	// Arrayposition entspricht dem absoluten Druck. Z.B. 1.00bara => 0.00bar Überdruck => Arrayposition 100
	R407cDew: ARRAY [0..5100] OF INT := [-1006,-937,-894,-862,-835,-813,-794,-777,-762,-748,-735,-723,-712,-702,-692,-683,-674,-666,-658,-650,-643,-636,-629,-622,-616,-610,-604,-598,-593,-587,-582,-577,-572,-567,-562,-557,-553,-548,-544,-540,-535,-531,-527,-523,-519,-515,-512,-508,-504,-501,-497,-494,-490,-487,-484,-480,-477,-474,-471,-468,-465,-462,-459,-456,-453,-450,-447,-445,-442,-439,-436,-434,-431,-428,-426,-423,-421,-418,-416,-413,-411,-409,-406,-404,-402,-399,-397,-395,-392,-390,-388,-386,-384,-382,-379,-377,-375,-373,-371,-369,-367,-365,-363,-361,-359,-357,-355,-353,-351,-349,-347,-346,-344,-342,-340,-338,-336,-335,-333,-331,-329,-328,-326,-324,-322,-321,-319,-317,-316,-314,-312,-311,-309,-307,-306,-304,-303,-301,-300,-298,-296,-295,-293,-292,-290,-289,-287,-286,-284,-283,-281,-280,-278,-277,-275,-274,-273,-271,-270,-268,-267,-266,-264,-263,-261,-260,-259,-257,-256,-255,-253,-252,-251,-249,-248,-247,-245,-244,-243,-241,-240,-239,-238,-236,-235,-234,-233,-231,-230,-229,-228,-226,-225,-224,-223,-222,-220,-219,-218,-217,-216,-215,-213,-212,-211,-210,-209,-208,-206,-205,-204,-203,-202,-201,-200,-199,-197,-196,-195,-194,-193,-192,-191,-190,-189,-188,-187,-185,-184,-183,-182,-181,-180,-179,-178,-177,-176,-175,-174,-173,-172,-171,-170,-169,-168,-167,-166,-165,-164,-163,-162,-161,-160,-159,-158,-157,-156,-155,-154,-153,-152,-151,-150,-149,-148,-147,-146,-145,-145,-144,-143,-142,-141,-140,-139,-138,-137,-136,-135,-134,-133,-133,-132,-131,-130,-129,-128,-127,-126,-125,-124,-124,-123,-122,-121,-120,-119,-118,-118,-117,-116,-115,-114,-113,-112,-112,-111,-110,-109,-108,-107,-106,-106,-105,-104,-103,-102,-101,-101,-100,-99,-98,-97,-97,-96,-95,-94,-93,-93,-92,-91,-90,-89,-89,-88,-87,-86,-85,-85,-84,-83,-82,-81,-81,-80,-79,-78,-78,-77,-76,-75,-75,-74,-73,-72,-71,-71,-70,-69,-68,-68,-67,-66,-65,-65,-64,-63,-63,-62,-61,-60,-60,-59,-58,-57,-57,-56,-55,-55,-54,-53,-52,-52,-51,-50,-50,-49,-48,-47,-47,-46,-45,-45,-44,-43,-42,-42,-41,-40,-40,-39,-38,-38,-37,-36,-36,-35,-34,-34,-33,-32,-32,-31,-30,-29,-29,-28,-27,-27,-26,-25,-25,-24,-23,-23,-22,-22,-21,-20,-20,-19,-18,-18,-17,-16,-16,-15,-14,-14,-13,-12,-12,-11,-11,-10,-9,-9,-8,-7,-7,-6,-5,-5,-4,-4,-3,-2,-2,-1,0,0,1,1,2,3,3,4,4,5,6,6,7,8,8,9,9,10,11,11,12,12,13,14,14,15,15,16,17,17,18,18,19,20,20,21,21,22,22,23,24,24,25,25,26,27,27,28,28,29,29,30,31,31,32,32,33,33,34,35,35,36,36,37,37,38,38,39,40,40,41,41,42,42,43,43,44,45,45,46,46,47,47,48,48,49,50,50,51,51,52,52,53,53,54,54,55,55,56,57,57,58,58,59,59,60,60,61,61,62,62,63,63,64,64,65,66,66,67,67,68,68,69,69,70,70,71,71,72,72,73,73,74,74,75,75,76,76,77,77,78,78,79,79,80,80,81,81,82,82,83,83,84,84,85,85,86,86,87,87,88,88,89,89,90,90,91,91,92,92,93,93,94,94,95,95,96,96,97,97,98,98,99,99,100,100,101,101,101,102,102,103,103,104,104,105,105,106,106,107,107,108,108,109,109,110,110,110,111,111,112,112,113,113,114,114,115,115,116,116,117,117,117,118,118,119,119,120,120,121,121,122,122,122,123,123,124,124,125,125,126,126,127,127,127,128,128,129,129,130,130,131,131,131,132,132,133,133,134,134,135,135,135,136,136,137,137,138,138,139,139,139,140,140,141,141,142,142,142,143,143,144,144,145,145,145,146,146,147,147,148,148,148,149,149,150,150,151,151,151,152,152,153,153,154,154,154,155,155,156,156,156,157,157,158,158,159,159,159,160,160,161,161,161,162,162,163,163,164,164,164,165,165,166,166,166,167,167,168,168,168,169,169,170,170,170,171,171,172,172,173,173,173,174,174,175,175,175,176,176,177,177,177,178,178,179,179,179,180,180,181,181,181,182,182,182,183,183,184,184,184,185,185,186,186,186,187,187,188,188,188,189,189,190,190,190,191,191,191,192,192,193,193,193,194,194,195,195,195,196,196,196,197,197,198,198,198,199,199,199,200,200,201,201,201,202,202,203,203,203,204,204,204,205,205,206,206,206,207,207,207,208,208,209,209,209,210,210,210,211,211,211,212,212,213,213,213,214,214,214,215,215,216,216,216,217,217,217,218,218,218,219,219,220,220,220,221,221,221,222,222,222,223,223,223,224,224,225,225,225,226,226,226,227,227,227,228,228,228,229,229,230,230,230,231,231,231,232,232,232,233,233,233,234,234,234,235,235,236,236,236,237,237,237,238,238,238,239,239,239,240,240,240,241,241,241,242,242,242,243,243,244,244,244,245,245,245,246,246,246,247,247,247,248,248,248,249,249,249,250,250,250,251,251,251,252,252,252,253,253,253,254,254,254,255,255,255,256,256,256,257,257,257,258,258,258,259,259,259,260,260,260,261,261,261,262,262,262,263,263,263,264,264,264,265,265,265,266,266,266,267,267,267,268,268,268,269,269,269,270,270,270,271,271,271,272,272,272,272,273,273,273,274,274,274,275,275,275,276,276,276,277,277,277,278,278,278,279,279,279,280,280,280,280,281,281,281,282,282,282,283,283,283,284,284,284,285,285,285,286,286,286,286,287,287,287,288,288,288,289,289,289,290,290,290,291,291,291,291,292,292,292,293,293,293,294,294,294,295,295,295,295,296,296,296,297,297,297,298,298,298,299,299,299,299,300,300,300,301,301,301,302,302,302,302,303,303,303,304,304,304,305,305,305,305,306,306,306,307,307,307,308,308,308,308,309,309,309,310,310,310,311,311,311,311,312,312,312,313,313,313,314,314,314,314,315,315,315,316,316,316,316,317,317,317,318,318,318,319,319,319,319,320,320,320,321,321,321,321,322,322,322,323,323,323,323,324,324,324,325,325,325,325,326,326,326,327,327,327,328,328,328,328,329,329,329,330,330,330,330,331,331,331,332,332,332,332,333,333,333,334,334,334,334,335,335,335,335,336,336,336,337,337,337,337,338,338,338,339,339,339,339,340,340,340,341,341,341,341,342,342,342,342,343,343,343,344,344,344,344,345,345,345,346,346,346,346,347,347,347,347,348,348,348,349,349,349,349,350,350,350,350,351,351,351,352,352,352,352,353,353,353,353,354,354,354,355,355,355,355,356,356,356,356,357,357,357,358,358,358,358,359,359,359,359,360,360,360,361,361,361,361,362,362,362,362,363,363,363,363,364,364,364,365,365,365,365,366,366,366,366,367,367,367,367,368,368,368,368,369,369,369,370,370,370,370,371,371,371,371,372,372,372,372,373,373,373,373,374,374,374,375,375,375,375,376,376,376,376,377,377,377,377,378,378,378,378,379,379,379,379,380,380,380,380,381,381,381,382,382,382,382,383,383,383,383,384,384,384,384,385,385,385,385,386,386,386,386,387,387,387,387,388,388,388,388,389,389,389,389,390,390,390,390,391,391,391,391,392,392,392,392,393,393,393,393,394,394,394,394,395,395,395,395,396,396,396,396,397,397,397,397,398,398,398,398,399,399,399,399,400,400,400,400,401,401,401,401,402,402,402,402,403,403,403,403,404,404,404,404,405,405,405,405,406,406,406,406,407,407,407,407,408,408,408,408,409,409,409,409,409,410,410,410,410,411,411,411,411,412,412,412,412,413,413,413,413,414,414,414,414,415,415,415,415,416,416,416,416,416,417,417,417,417,418,418,418,418,419,419,419,419,420,420,420,420,421,421,421,421,421,422,422,422,422,423,423,423,423,424,424,424,424,425,425,425,425,426,426,426,426,426,427,427,427,427,428,428,428,428,429,429,429,429,429,430,430,430,430,431,431,431,431,432,432,432,432,433,433,433,433,433,434,434,434,434,435,435,435,435,436,436,436,436,436,437,437,437,437,438,438,438,438,439,439,439,439,439,440,440,440,440,441,441,441,441,441,442,442,442,442,443,443,443,443,444,444,444,444,444,445,445,445,445,446,446,446,446,446,447,447,447,447,448,448,448,448,449,449,449,449,449,450,450,450,450,451,451,451,451,451,452,452,452,452,453,453,453,453,453,454,454,454,454,455,455,455,455,455,456,456,456,456,457,457,457,457,457,458,458,458,458,459,459,459,459,459,460,460,460,460,461,461,461,461,461,462,462,462,462,462,463,463,463,463,464,464,464,464,464,465,465,465,465,466,466,466,466,466,467,467,467,467,467,468,468,468,468,469,469,469,469,469,470,470,470,470,471,471,471,471,471,472,472,472,472,472,473,473,473,473,474,474,474,474,474,475,475,475,475,475,476,476,476,476,477,477,477,477,477,478,478,478,478,478,479,479,479,479,479,480,480,480,480,481,481,481,481,481,482,482,482,482,482,483,483,483,483,484,484,484,484,484,485,485,485,485,485,486,486,486,486,486,487,487,487,487,487,488,488,488,488,489,489,489,489,489,490,490,490,490,490,491,491,491,491,491,492,492,492,492,492,493,493,493,493,493,494,494,494,494,495,495,495,495,495,496,496,496,496,496,497,497,497,497,497,498,498,498,498,498,499,499,499,499,499,500,500,500,500,500,501,501,501,501,501,502,502,502,502,502,503,503,503,503,504,504,504,504,504,505,505,505,505,505,506,506,506,506,506,507,507,507,507,507,508,508,508,508,508,509,509,509,509,509,510,510,510,510,510,511,511,511,511,511,512,512,512,512,512,513,513,513,513,513,514,514,514,514,514,515,515,515,515,515,515,516,516,516,516,516,517,517,517,517,517,518,518,518,518,518,519,519,519,519,519,520,520,520,520,520,521,521,521,521,521,522,522,522,522,522,523,523,523,523,523,524,524,524,524,524,525,525,525,525,525,525,526,526,526,526,526,527,527,527,527,527,528,528,528,528,528,529,529,529,529,529,530,530,530,530,530,530,531,531,531,531,531,532,532,532,532,532,533,533,533,533,533,534,534,534,534,534,535,535,535,535,535,535,536,536,536,536,536,537,537,537,537,537,538,538,538,538,538,539,539,539,539,539,539,540,540,540,540,540,541,541,541,541,541,542,542,542,542,542,542,543,543,543,543,543,544,544,544,544,544,545,545,545,545,545,545,546,546,546,546,546,547,547,547,547,547,548,548,548,548,548,548,549,549,549,549,549,550,550,550,550,550,550,551,551,551,551,551,552,552,552,552,552,553,553,553,553,553,553,554,554,554,554,554,555,555,555,555,555,555,556,556,556,556,556,557,557,557,557,557,557,558,558,558,558,558,559,559,559,559,559,559,560,560,560,560,560,561,561,561,561,561,561,562,562,562,562,562,563,563,563,563,563,563,564,564,564,564,564,565,565,565,565,565,565,566,566,566,566,566,567,567,567,567,567,567,568,568,568,568,568,568,569,569,569,569,569,570,570,570,570,570,570,571,571,571,571,571,572,572,572,572,572,572,573,573,573,573,573,573,574,574,574,574,574,575,575,575,575,575,575,576,576,576,576,576,576,577,577,577,577,577,578,578,578,578,578,578,579,579,579,579,579,579,580,580,580,580,580,580,581,581,581,581,581,582,582,582,582,582,582,583,583,583,583,583,583,584,584,584,584,584,585,585,585,585,585,585,586,586,586,586,586,586,587,587,587,587,587,587,588,588,588,588,588,588,589,589,589,589,589,590,590,590,590,590,590,591,591,591,591,591,591,592,592,592,592,592,592,593,593,593,593,593,593,594,594,594,594,594,594,595,595,595,595,595,595,596,596,596,596,596,597,597,597,597,597,597,598,598,598,598,598,598,599,599,599,599,599,599,600,600,600,600,600,600,601,601,601,601,601,601,602,602,602,602,602,602,603,603,603,603,603,603,604,604,604,604,604,604,605,605,605,605,605,605,606,606,606,606,606,606,607,607,607,607,607,607,608,608,608,608,608,608,609,609,609,609,609,609,610,610,610,610,610,610,611,611,611,611,611,611,612,612,612,612,612,612,613,613,613,613,613,613,614,614,614,614,614,614,615,615,615,615,615,615,615,616,616,616,616,616,616,617,617,617,617,617,617,618,618,618,618,618,618,619,619,619,619,619,619,620,620,620,620,620,620,621,621,621,621,621,621,622,622,622,622,622,622,622,623,623,623,623,623,623,624,624,624,624,624,624,625,625,625,625,625,625,626,626,626,626,626,626,627,627,627,627,627,627,627,628,628,628,628,628,628,629,629,629,629,629,629,630,630,630,630,630,630,630,631,631,631,631,631,631,632,632,632,632,632,632,633,633,633,633,633,633,634,634,634,634,634,634,634,635,635,635,635,635,635,636,636,636,636,636,636,637,637,637,637,637,637,637,638,638,638,638,638,638,639,639,639,639,639,639,639,640,640,640,640,640,640,641,641,641,641,641,641,642,642,642,642,642,642,642,643,643,643,643,643,643,644,644,644,644,644,644,644,645,645,645,645,645,645,646,646,646,646,646,646,646,647,647,647,647,647,647,648,648,648,648,648,648,648,649,649,649,649,649,649,650,650,650,650,650,650,650,651,651,651,651,651,651,652,652,652,652,652,652,652,653,653,653,653,653,653,654,654,654,654,654,654,654,655,655,655,655,655,655,655,656,656,656,656,656,656,657,657,657,657,657,657,657,658,658,658,658,658,658,659,659,659,659,659,659,659,660,660,660,660,660,660,660,661,661,661,661,661,661,662,662,662,662,662,662,662,663,663,663,663,663,663,663,664,664,664,664,664,664,665,665,665,665,665,665,665,666,666,666,666,666,666,666,667,667,667,667,667,667,667,668,668,668,668,668,668,669,669,669,669,669,669,669,670,670,670,670,670,670,670,671,671,671,671,671,671,671,672,672,672,672,672,672,673,673,673,673,673,673,673,674,674,674,674,674,674,674,675,675,675,675,675,675,675,676,676,676,676,676,676,676,677,677,677,677,677,677,677,678,678,678,678,678,678,678,679,679,679,679,679,679,680,680,680,680,680,680,680,681,681,681,681,681,681,681,682,682,682,682,682,682,682,683,683,683,683,683,683,683,684,684,684,684,684,684,684,685,685,685,685,685,685,685,686,686,686,686,686,686,686,687,687,687,687,687,687,687,688,688,688,688,688,688,688,689,689,689,689,689,689,689,690,690,690,690,690,690,690,691,691,691,691,691,691,691,692,692,692,692,692,692,692,693,693,693,693,693,693,693,694,694,694,694,694,694,694,695,695,695,695,695,695,695,695,696,696,696,696,696,696,696,697,697,697,697,697,697,697,698,698,698,698,698,698,698,699,699,699,699,699,699,699,700,700,700,700,700,700,700,701,701,701,701,701,701,701,701,702,702,702,702,702,702,702,703,703,703,703,703,703,703,704,704,704,704,704,704,704,705,705,705,705,705,705,705,705,706,706,706,706,706,706,706,707,707,707,707,707,707,707,708,708,708,708,708,708,708,709,709,709,709,709,709,709,709,710,710,710,710,710,710,710,711,711,711,711,711,711,711,712,712,712,712,712,712,712,712,713,713,713,713,713,713,713,714,714,714,714,714,714,714,715,715,715,715,715,715,715,715,716,716,716,716,716,716,716,717,717,717,717,717,717,717,717,718,718,718,718,718,718,718,719,719,719,719,719,719,719,719,720,720,720,720,720,720,720,721,721,721,721,721,721,721,721,722,722,722,722,722,722,722,723,723,723,723,723,723,723,723,724,724,724,724,724,724,724,725,725,725,725,725,725,725,725,726,726,726,726,726,726,726,727,727,727,727,727,727,727,727,728,728,728,728,728,728,728,729,729,729,729,729,729,729,729,730,730,730,730,730,730,730,730,731,731,731,731,731,731,731,732,732,732,732,732,732,732,732,733,733,733,733,733,733,733,733,734,734,734,734,734,734,734,735,735,735,735,735,735,735,735,736,736,736,736,736,736,736,736,737,737,737,737,737,737,737,738,738,738,738,738,738,738,738,739,739,739,739,739,739,739,739,740,740,740,740,740,740,740,740,741,741,741,741,741,741,741,741,742,742,742,742,742,742,742,743,743,743,743,743,743,743,743,744,744,744,744,744,744,744,744,745,745,745,745,745,745,745,745,746,746,746,746,746,746,746,746,747,747,747,747,747,747,747,747,748,748,748,748,748,748,748,748,749,749,749,749,749,749,749,749,750,750,750,750,750,750,750,750,751,751,751,751,751,751,751,752,752,752,752,752,752,752,752,753,753,753,753,753,753,753,753,754,754,754,754,754,754,754,754,755,755,755,755,755,755,755,755,755,756,756,756,756,756,756,756,756,757,757,757,757,757,757,757,757,758,758,758,758,758,758,758,758,759,759,759,759,759,759,759,759,760,760,760,760,760,760,760,760,761,761,761,761,761,761,761,761,762,762,762,762,762,762,762,762,763,763,763,763,763,763,763,763,764,764,764,764,764,764,764,764,764,765,765,765,765,765,765,765,765,766,766,766,766,766,766,766,766,767,767,767,767,767,767,767,767,768,768,768,768,768,768,768,768,768,769,769,769,769,769,769,769,769,770,770,770,770,770,770,770,770,771,771,771,771,771,771,771,771,771,772,772,772,772,772,772,772,772,773,773,773,773,773,773,773,773,774,774,774,774,774,774,774,774,774,775,775,775,775,775,775,775,775,776,776,776,776,776,776,776,776,777,777,777,777,777,777,777,777,777,778,778,778,778,778,778,778,778,779,779,779,779,779,779,779,779,779,780,780,780,780,780,780,780,780,781,781,781,781,781,781,781,781,781,782,782,782,782,782,782,782,782,783,783,783,783,783,783,783,783,783,784,784,784,784,784,784,784,784,784,785,785,785,785,785,785,785,785,786,786,786,786,786,786,786,786,786,787,787,787,787,787,787,787,787,788,788,788,788,788,788,788,788,788,789,789,789,789,789,789,789,789,789,790,790,790,790,790,790,790,790,791,791,791,791,791,791,791,791,791,792,792,792,792,792,792,792,792,792,793,793,793,793,793,793,793,793,793,794,794,794,794,794,794,794,794,795,795,795,795,795,795,795,795,795,796,796,796,796,796,796,796,796,796,797,797,797,797,797,797,797,797,797,798,798,798,798,798,798,798,798,798,799,799,799,799,799,799,799,799,799,800,800,800,800,800,800,800,800,800,801,801,801,801,801,801,801,801,801,802,802,802,802,802,802,802,802,802,803,803,803,803,803,803,803,803,803,804,804,804,804,804,804,804,804,804,805,805,805,805,805,805,805,805,805,806,806,806,806,806,806,806,806,806,807,807,807,807,807,807,807,807,807,808,808,808,808,808,808,808,808,808,809,809,809,809,809,809,809,809,809,810,810,810,810,810,810,810,810,810,811,811,811,811,811,811,811,811,811,811,812,812,812,812,812,812,812,812,812,813,813,813,813,813,813,813,813,813,814,814,814,814,814,814,814,814,814,815,815,815,815,815,815,815,815,815,815,816,816,816,816,816,816,816,816,816,817,817,817,817,817,817,817,817,817,818,818,818,818,818,818,818,818,818,818,819,819,819,819,819,819,819,819,819,820,820,820,820,820,820,820,820,820,820,821,821,821,821,821,821,821,821,821,822,822,822,822,822,822,822,822,822,822,823,823,823,823,823,823,823,823,823,824,824];

END_VAR

// Globale Variablen/SW_ALZ
{attribute 'qualified_only'}
VAR_GLOBAL
	Bitzer_Scroll_R410a: SW_Einsatzgrenzen := (f_SW_EG_MinVerd := -30, f_SW_EG_MaxVerd := 21, f_SW_EG_MinKond := 25, f_SW_EG_MaxKond := 65, f_SW_EG_BVerd := 12.5, f_SW_EG_BKond := 25, f_SW_EG_CKond := 38, f_SW_EG_DKond := 65, f_SW_EG_EVerd := 21, f_SW_EG_FVerd := 0, f_SW_EG_GKond := 32, f_SW_Max_HeissgasTemp := 120);
END_VAR

// Globale Variablen/Visu
{attribute 'qualified_only'}
VAR_GLOBAL
	i_Frame_Index:INT;
	i_Verschiebung_Horizontal:INT;
	i_Verschiebung_Vertikal:INT;
	x_Quittieren: BOOL;
END_VAR

// Version/Global_Version
{attribute 'TcGenerated'}
// This function has been automatically generated from the project information.
VAR_GLOBAL CONSTANT
	{attribute 'const_non_replaced'}
	{attribute 'linkalways'}
	stLibVersion_GWP_Library : ST_LibVersion := (iMajor := 17, iMinor := 9, iBuild := 1, iRevision := 0, sVersion := '17.9.1');
END_VAR

// Allgemein/Alarm
(*Alarmblock, welcher ein digitaler Ausgang high setzt wenn mind. Ein Alarm anstehend ist und ebenfalls noch die Selbsthaltung der Alarme
*)
FUNCTION_BLOCK Alarm
(*
Versionsverlauf: 
Version		|Autor	|Bemerkung
------------------------------------------------------------------------------------------------------------ 
17.06.00	|Shgb	|erste Freigabe 
17.08.00	|LeaF	|Freigabe

*)
VAR_INPUT
	x_AL1:BOOL;//Alarmeingang 1-16
	x_AL2:BOOL;
	x_AL3:BOOL;
	x_AL4:BOOL;
	x_AL5:BOOL;
	x_AL6:BOOL;
	x_AL7:BOOL;
	x_AL8:BOOL;
	x_AL9:BOOL;
	x_AL10:BOOL;
END_VAR
VAR_OUTPUT	
	x_Aus:BOOL;//Allgemeiner Alarm
	x_AL_1:BOOL;//Alarmausgang 1-16
	x_AL_2:BOOL;
	x_AL_3:BOOL;
	x_AL_4:BOOL;
	x_AL_5:BOOL;
	x_AL_6:BOOL;
	x_AL_7:BOOL;
	x_AL_8:BOOL;
	x_AL_9:BOOL;
	x_AL_10:BOOL;
END_VAR
VAR Persistent
	ax_AL :ARRAY [1..10] OF BOOL;
	ax_Speicher :ARRAY [1..10] OF BOOL;
	i_Arraypos:INT;
	as_Liste: ARRAY [1..10] OF STRING;
END_VAR

//Array füllen
	ax_AL[1]:=x_AL1;
	ax_AL[2]:=x_AL2;
	ax_AL[3]:=x_AL3;
	ax_AL[4]:=x_AL4;
	ax_AL[5]:=x_AL5;
	ax_AL[6]:=x_AL6;
	ax_AL[7]:=x_AL7;
	ax_AL[8]:=x_AL8;
	ax_AL[9]:=x_AL9;
	ax_AL[10]:=x_AL10;
	
//Quittieren
	IF Globale_Variablen.x_Quittieren THEN
		FOR i_Arraypos:=1 TO 10 DO
			ax_Speicher[i_Arraypos]:=FALSE;
		END_FOR
	END_IF

//Alarme Setzen
	FOR i_Arraypos:=1 TO 10 DO
		IF ax_AL[i_Arraypos] THEN
			ax_Speicher[i_Arraypos]:=TRUE;
		END_IF
	END_FOR

//Ausgäne setzen
	x_AL_1:=ax_Speicher[1];
	x_AL_2:=ax_Speicher[2];
	x_AL_3:=ax_Speicher[3];
	x_AL_4:=ax_Speicher[4];
	x_AL_5:=ax_Speicher[5];
	x_AL_6:=ax_Speicher[6];
	x_AL_7:=ax_Speicher[7];
	x_AL_8:=ax_Speicher[8];
	x_AL_9:=ax_Speicher[9];
	x_AL_10:=ax_Speicher[10];
	
	x_Aus:=x_al_1 OR 
			x_al_2 OR 
			x_al_3 OR 
			x_al_4 OR
			x_al_5 OR
			x_al_6 OR
			x_al_7 OR
			x_al_8 OR
			x_al_9 OR
			x_al_10;

END_FUNCTION_BLOCK

// Allgemein/COUNT
(*Je nachdem wieviele digitale Eingänge true sind, wird er analoge Ausgang hochgezählt. Ist kein Eingang auf true, bleibt der Ausgang auf 0.
Der Counter ist auf max. 8 digitale Eingänge ausgelegt.
*)
FUNCTION_BLOCK COUNT
(*
Versionsverlauf: 
Version		|Autor	|Bemerkung
------------------------------------------------------------------------------------------------------------ 
17.05.00	|KuzR	|erste Freigabe  
17.08.00	|LeaF	|Freigabe

*)
VAR_INPUT	
	x_Ein_1:BOOL;//8 Digitale Eingänge
	x_Ein_2:BOOL;
	x_Ein_3:BOOL;
	x_Ein_4:BOOL;
	x_Ein_5:BOOL;
	x_Ein_6:BOOL;
	x_Ein_7:BOOL;
	x_Ein_8:BOOL;
END_VAR
VAR_OUTPUT
	i_Aus:Int;//Ausganng in Int
END_VAR
VAR	
END_VAR

	i_Aus:=0;
// Ausgang zählt hoch, wenn Eingang true ist
	IF x_Ein_1 THEN
		i_Aus:=i_Aus+1;
	END_IF
	
	IF x_Ein_2 THEN
		i_Aus:=i_Aus+1;
	END_IF
	
	IF x_Ein_3 THEN
		i_Aus:=i_Aus+1;
	END_IF
	
	IF x_Ein_4 THEN
		i_Aus:=i_Aus+1;
	END_IF
	
	IF x_Ein_5 THEN
		i_Aus:=i_Aus+1;
	END_IF
	
	IF x_Ein_6 THEN
		i_Aus:=i_Aus+1;
	END_IF
	
	IF x_Ein_7 THEN
		i_Aus:=i_Aus+1;
	END_IF
	
	IF x_Ein_8 THEN
		i_Aus:=i_Aus+1;
	END_IF

END_FUNCTION_BLOCK

// Allgemein/MUX_B
(*Anhand von 4 digitalen Eingängen wird entschieden, welcher von 4 analogen Werten (Real) auf den analogen Ausgang (Real) geschrieben wird.
Der kleinere Eingang hat immer Priorität für das Schreiben des Ausganges. Wenn keine Eingänge auf true sind, dann Augang auf 0.

*)
FUNCTION_BLOCK MUX_B
(*
Versionsverlauf: 
Version		|Autor	|Bemerkung
------------------------------------------------------------------------------------------------------------ 
17.06.00	|KuzR	|erste Freigabe  
17.08.00	|LeaF	|Freigabe

*)
VAR_INPUT
	f_Ein_1:REAL;//Eingangswerte 1-4 in Real
	f_Ein_2:REAL;
	f_Ein_3:REAL;
	f_Ein_4:REAL;
	x_Ein_1:BOOL;//Digitaler Eingang 1
	x_Ein_2:BOOL;//Digitaler Eingang 2
	x_Ein_3:BOOL;//Digitaler Eingang 3
	x_Ein_4:BOOL;//Digitaler Eingang 4
END_VAR
VAR_OUTPUT
	f_Aus:REAL;//Ausgang in Real
END_VAR
VAR
END_VAR

	f_Aus:=0;
//Wenn 1.Eingang True, dann Wert1
	IF x_Ein_1  THEN
		f_Aus := f_Ein_1;		
//Ansonsen wird beim Ausgang Wert zwei geschrieben
	ELSIF x_Ein_2 THEN
		f_Aus := f_Ein_2;		
	ELSIF x_Ein_3 THEN
		f_Aus := f_Ein_3;		
	ELSIF x_Ein_4 THEN
		f_Aus := f_Ein_4;							
	END_IF

END_FUNCTION_BLOCK

// Allgemein/MUX_D_INT
(*Anhand von 3 analogen Eingangswerten (Integer)wird mit dem i_Sel entschieden, welcher von den 3 Eingängen auf den analogen Ausgang (Integer) geschrieben wird.
*)
FUNCTION_BLOCK MUX_D_INT
(*
Versionsverlauf: 
Version		|Autor	|Bemerkung
------------------------------------------------------------------------------------------------------------ 
17.05.00	|KuzR	|erste Freigabe  
17.08.00	|LeaF	|Freigabe

*)
VAR_INPUT
	i_Ein_1:INT;//Eingangswert 1 als Int
	i_Ein_2:INT;//Eingangswert 2 als Int
	i_Ein_3:INT; //Eingangswert 3 als Int
	i_Sel:INT;// Auswahl Selector
	
END_VAR
VAR_OUTPUT
	i_Aus:INT;//Ausgang als Int
END_VAR
VAR
END_VAR

//Mit Select Auswählen, welcher Eingang auf Ausgang geschrieben wird
	CASE i_sel OF
		1: i_Aus:= i_Ein_1;
		2: i_Aus:= i_Ein_2;
		3: i_Aus:= i_Ein_3;
	ELSE	
//Wenn Select <3 oder >0, dann Ausgang 0
		i_Aus:=0;
	END_CASE

END_FUNCTION_BLOCK

// Allgemein/MUX_D_REAL
(*Anhand von 3 analogen Eingangswerten (Real)wird mit dem i_Sel entschieden, welcher von den 3 Eingängen auf den analogen Ausgang (Real) geschrieben wird.
*)
FUNCTION_BLOCK MUX_D_REAL
(*
Versionsverlauf: 
Version		|Autor	|Bemerkung
------------------------------------------------------------------------------------------------------------ 
17.06.00	|ShgB	|erste Freigabe  
17.08.00	|LeaF	|Freigabe

*)
VAR_INPUT
	f_Ein_1:REAL;//Eingangswert 1 als Real
	f_Ein_2:REAL;//Eingangswert 2 als Real
	f_Ein_3:REAL;//Eingangswert 3 als Real
	i_Sel:INT;// Auswahl Selector
	
END_VAR
VAR_OUTPUT
	f_Aus:REAL;//Ausgang in Real
END_VAR
VAR
END_VAR

//Mit Select Auswählen, welcher Eingang auf Ausgang geschrieben wird
	CASE i_sel OF
		1: f_Aus:= f_Ein_1;
		2: f_Aus:= f_Ein_2;
		3: f_Aus:= f_Ein_3;
	ELSE
		
//Wenn Select <0 oder >3, dann Ausgang 0
		f_Aus:=0;
	END_CASE

END_FUNCTION_BLOCK

// Allgemein/NULL
(*Wenn der analoge Eingang (Real) genau 0 ist, wird der digitale Ausgang auf true gesetzt, ansonsten auf false.
*)
FUNCTION_BLOCK NULL
(*
Versionsverlauf: 
Version		|Autor	|Bemerkung
------------------------------------------------------------------------------------------------------------ 
17.06.00	|KuzR	|erste Freigabe  
17.08.00	|LeaF	|Freigabe

*)
VAR_INPUT
	i_Ein:REAL;//Eingangswert in Real
END_VAR
VAR_OUTPUT
	x_Aus:BOOL;//Digitaler Ausgang
END_VAR
VAR
END_VAR

//Wenn 0 gleich Ausgang true, ansonsten false
	x_Aus:=i_Ein =0;

END_FUNCTION_BLOCK

// Allgemein/SWITCH_INT
(*Ist der digitale Eingang auf false, wird der erste analoge Eingangswert (Int) in den analogen Ausgang (Int) geschrieben. 
Ist der digitale Eingang auf true, wird der zweite analoge Eingangswert (Int) in den analogen Ausgang (Int) geschrieben.
*)
FUNCTION_BLOCK SWITCH_INT
(*
Versionsverlauf: 
Version		|Autor	|Bemerkung
------------------------------------------------------------------------------------------------------------ 
17.05.00	|KuzR	|erste Freigabe  
17.08.00	|LeaF	|Freigabe

*)
VAR_INPUT
	x_Ein:BOOL;//Digitaler Eingang
	i_Ein_1:INT;//Analoger Eingangswert 1 als Int
	i_Ein_2:INT;//Analoger Eingangswert 2 als Int
END_VAR
VAR_OUTPUT
	i_Aus:INT;//Analoger Ausgangswert als Int
END_VAR
VAR	
END_VAR

	IF x_Ein THEN		
//Wenn Eingang True, Wert_2 in Ausgang
		i_Aus:= i_Ein_2;	
	ELSE	
//Wenn Eingang false, Wert_1 in Ausgang
		i_Aus:= i_Ein_1;
	END_IF

END_FUNCTION_BLOCK

// Allgemein/SWITCH_REAL
(*Ist der digitale Eingang auf false, wird der erste analoge Eingangswert (Real) in den analogen Ausgang (Real) geschrieben. 
Ist der digitale Eingang auf true, wird der zweite analoge Eingangswert (Real) in den analogen Ausgang (Real) geschrieben.
*)
FUNCTION_BLOCK SWITCH_REAL
(*
Versionsverlauf: 
Version		|Autor	|Bemerkung
------------------------------------------------------------------------------------------------------------ 
17.05.00	|KuzR	|erste Freigabe  
17.08.00	|LeaF	|Freigabe

*)
VAR_INPUT
	x_Ein:BOOL;//Digitaler Eingang
	f_Ein_1:REAL;//Analoger Eingangswert 1 als Real
	f_Ein_2	:REAL;//Analoger Eingangswert 2 als Real
END_VAR
VAR_OUTPUT
	f_Aus:REAL;//Analoger Ausgangswert als Real
END_VAR
VAR	
END_VAR

	IF x_Ein THEN		
//Wenn Eingang True, Wert_2 in Ausgang
		f_Aus:= f_Ein_2;	
	ELSE	
//Wenn Eingang false, Wert_1 in Ausgang
		f_Aus:= f_Ein_1;
	END_IF

END_FUNCTION_BLOCK

// Allgemein/Toggle
(*Mit einer positiven Flanke auf den x_Toggle Eingang wird der Wert des Ausgangs x_Aus zwischen FALSE und TRUE gwechselt.
Mit dem x_Reset Eingang kann der Ausgang auf FALSE geschrieben werden. 
*)
FUNCTION_BLOCK Toggle
(*
Versionsverlauf: 
Version		|Autor	|Bemerkung
------------------------------------------------------------------------------------------------------------ 
17.06.00	|Shgb	|erste Freigabe  
17.08.00	|LeaF	|Freigabe

*)
VAR_INPUT
	x_Toggle:BOOL;//Wechselt den Wert des Ausgangs bei einer positiven Flanke
	x_Reset:BOOL;//Setzt den Ausgang auf FALSE
END_VAR
VAR_OUTPUT
	x_Aus:BOOL;//Ausgang
END_VAR
VAR PERSISTENT
	x_Speicher: BOOL;
END_VAR
VAR
	x_Flanke:BOOL;
END_VAR

//Toggle mit Flankenerkennung
	IF x_Toggle AND NOT x_Flanke THEN
		x_Speicher:= NOT x_Speicher;
	END_IF
	x_Flanke:=x_Toggle;

//Reset
	IF x_Reset THEN
		x_Speicher:=FALSE;
	END_IF
	
//Ausgang schreiben
	x_Aus:=x_Speicher;

END_FUNCTION_BLOCK

// Converters/Converter2Punkt
(*Der Eingang f_Ein wird anhand des Bereiches von f_Ein_Min f_Ein_Max auf den Bereich f_Aus_Min und f_Aus_Max berechnet und auf den Ausgang f_Aus gegeben.
*)
FUNCTION_BLOCK Converter2Punkt
(*
Versionsverlauf: 
Version		|Autor	|Bemerkung
------------------------------------------------------------------------------------------------------------ 
17.06.00	|ShgB	|erste Freigabe 
17.06.01	|ShgB	|von Integer auf Real geändert 
17.08.00	|LeaF	|Freigabe	

*)
VAR_INPUT
	f_Ein:REAL;//Eingang
	f_Ein_Min:REAL;//Eingangsbereich Minimum
	f_Ein_Max:REAL;//Eingangsbereich Maximum
	f_Aus_Min:REAL;//Ausgangsbereich Minimum
	f_Aus_Max:REAL;//Ausgangsbereich Maximum
END_VAR
VAR_OUTPUT
	f_Aus:REAL;//Ausgang
END_VAR
VAR
END_VAR

IF f_Ein_Max-f_Ein_Min <> 0 THEN
	f_Aus:=(f_Aus_Max-f_Aus_Min)/(f_Ein_Max-f_Ein_Min)*(f_Ein-f_Ein_Min)+f_Aus_Min;
ELSE
	f_Aus:=f_Aus_Max;
END_IF

END_FUNCTION_BLOCK

// Math/Maximum
(*Gibt den grössten der angeschlossenen Werten aus.
*)
FUNCTION_BLOCK Maximum
(*
Versionsverlauf: 
Version		|Autor	|Bemerkung
------------------------------------------------------------------------------------------------------------ 
17.06.00	|Shgb	|erste Freigabe 
17.06.01	|ShgB	|von Integer auf Real geändert	 
17.08.00	|LeaF	|Freigabe

*)
VAR_INPUT
	f_Ein1 :REAL:=0.00001;//Wert 1
	f_Ein2 :REAL:=0.00001;//Wert 2
	f_Ein3 :REAL:=0.00001;//Wert 3
	f_Ein4 :REAL:=0.00001;//Wert 4
	f_Ein5 :REAL:=0.00001;//Wert 5
	f_Ein6 :REAL:=0.00001;//Wert 6
	f_Ein7 :REAL:=0.00001;//Wert 7
	f_Ein8 :REAL:=0.00001;//Wert 8
END_VAR
VAR_OUTPUT
	f_Aus:REAL;//Grösste Wert
END_VAR
VAR
	i_Arraypos:INT;
	af_Array: ARRAY [1..8] OF REAL;
END_VAR

// Werte in Array platzieren
	af_Array[1]:=f_Ein1;
	af_Array[2]:=f_Ein2;
	af_Array[3]:=f_Ein3;
	af_Array[4]:=f_Ein4;
	af_Array[5]:=f_Ein5;
	af_Array[6]:=f_Ein6;
	af_Array[7]:=f_Ein7;
	af_Array[8]:=f_Ein8;
	
//Zahlen die kleiner als 0 sind
	f_Aus := af_Array[1];	
	
//Auswertung der grössten Zahl
	FOR i_Arraypos:=2 TO 8 DO
		IF af_Array[i_Arraypos] >= f_Aus AND af_Array[i_Arraypos] <> 0.00001 THEN
			f_Aus := af_Array[i_Arraypos];
		END_IF
	END_FOR

END_FUNCTION_BLOCK

// Converters/Int_to_Druck
(*Der analoge Wert der Eingangskarte wird von einem 16 bit Integer in einen REAL Wert umgewandelt und ein Offset dazu addiert.
Standardmässig ist der Eingangsbereich von 0 - 32767 eingestellt. Sollte dieser nicht übereinstimmen kann der Bereich angepasst werden.
*)
FUNCTION_BLOCK Int_to_Druck
(*
Versionsverlauf: 
Version		|Autor	|Bemerkung
------------------------------------------------------------------------------------------------------------ 
17.06.00	|Shgb	|erste Freigabe  
17.08.00	|LeaF	|Freigabe

*)
VAR_INPUT
	i_Ein:INT;//Digitaler Eingangswert
END_VAR
VAR_INPUT PERSISTENT
	i_Ein_Min:INT:=0;//Eingangsbereich Minimum
	i_Ein_Max:INT:=32767;//Eingangsbereich Maximum
	f_Aus_Min:REAL;//Minimum des Drucktransmitters
	f_Aus_Max:REAL;//Maximum des Drucktransmitters
	f_Offset:REAL;//Offset der dazu addiert wird
END_VAR
VAR_OUTPUT
	f_Aus:REAL;//Druck im REAL Format
END_VAR
VAR//GUI Variablen
	f_GUI_Input:REAL;
END_VAR

IF i_Ein_Max-i_Ein_Min <> 0 THEN
	f_Aus:=(f_Aus_Max-f_Aus_Min)/(i_Ein_Max-i_Ein_Min)*(i_Ein-i_Ein_Min)+f_Aus_Min+f_Offset;
ELSE
	f_Aus:=f_Aus_Min;
END_IF

f_GUI_Input:=f_Aus-f_Offset;

END_FUNCTION_BLOCK

// Converters/Int_to_Temperature
(*Wandelt die Temperatur im INT Format, die von der Eingangskarte kommt, in eine Temperatur in REAL Format um und rechnet einen Offset dazu.
*)
FUNCTION_BLOCK Int_to_Temperature
(*
Versionsverlauf: 
Version		|Autor	|Bemerkung
------------------------------------------------------------------------------------------------------------ 
17.06.00	|Shgb	|erste Freigabe  
17.08.00	|LeaF	|Freigabe

*)
VAR_INPUT
	i_Ein:INT;//Temperatur von Karte
END_VAR
VAR_INPUT PERSISTENT
	f_Offset:REAL;//Offset der dazu addiert wird
END_VAR
VAR_OUTPUT
	f_Temperatur:REAL;//Ausgang REAL
END_VAR
VAR//GUI Variablen
	f_GUI_Input:REAL;
END_VAR

f_Temperatur:=i_Ein/10.0+f_Offset;
f_GUI_Input:=i_Ein/10.0;

END_FUNCTION_BLOCK

// Converters/Prozent_to_Int
(*Wandelt eine Prozentangabe vom Format REAL in eine Integer Zahl für die analoge Augangskarte um.
Standardmässig ist der Eingangsbereich von 0 - 32767 eingestellt. Sollte dieser nicht übereinstimmen kann der Bereich angepasst werden.
*)
FUNCTION_BLOCK Prozent_to_Int
(*
Versionsverlauf: 
Version		|Autor	|Bemerkung
------------------------------------------------------------------------------------------------------------ 
17.06.00	|Shgb	|erste Freigabe 
17.08.00	|LeaF	|Freigabe 

*)
VAR_INPUT
	f_Ein:REAL;//Eingang in Prozent
END_VAR
VAR_INPUT PERSISTENT
	i_Aus_Min:INT:=0;//Eingangsbereich Minimum
	i_Aus_Max:INT:=32767;//eingangsbereich Maximum
END_VAR
VAR_OUTPUT
	f_Aus:INT;//Ausgang
END_VAR
VAR
END_VAR

f_Aus:=real_to_int((i_Aus_Max-i_Aus_Min)*f_Ein/100.0);

END_FUNCTION_BLOCK

// Converters/Time_to_Timestruct
(*Wandelt die Eingangsvariable vom Typ TIME in ein TIMESTRUCT um.
*)
FUNCTION_BLOCK Time_to_Timestruct
(*
Versionsverlauf: 
Version		|Autor	|Bemerkung
------------------------------------------------------------------------------------------------------------ 
17.06.00	|Shgb	|erste Freigabe 	 
17.08.00	|LeaF	|Freigabe

*)
VAR_INPUT
	t_Ein:TIME;//Eingang
END_VAR
VAR_OUTPUT
	t_Aus:timestruct;//Ausgang
END_VAR
VAR
	OT:OTSTRUCT;
END_VAR

OT:=TIME_TO_OTSTRUCT(t_Ein);
t_Aus.wMilliseconds:=ot.wMilliseconds;
t_Aus.wSecond:=ot.wSecond;
t_Aus.wMinute:=ot.wMinute;
t_Aus.wHour:=ot.wHour;
t_Aus.wDay:=ot.wDay+ot.wWeek*7;

END_FUNCTION_BLOCK

// Converters/Timestruct_to_Time
(*Wandelt einen TIMESTRUCT in die Ausgangsvariable vom Typ TIME um.
*)
FUNCTION_BLOCK Timestruct_to_Time
(*
Versionsverlauf: 
Version		|Autor	|Bemerkung
------------------------------------------------------------------------------------------------------------ 
17.06.00	|Shgb	|erste Freigabe  
17.08.00	|LeaF	|Freigabe	

*)
VAR_INPUT
	t_Ein:timestruct;//Eingang
END_VAR
VAR_OUTPUT
	t_Aus:TIME;//Ausgang
END_VAR
VAR
END_VAR

t_Aus:=DINT_TO_TIME(t_Ein.wMilliseconds
					+ t_Ein.wSecond*1000
					+ t_Ein.wMinute*1000*60
					+ t_Ein.wHour*1000*60*60
					+ t_Ein.wDay*1000*60*60*24);

END_FUNCTION_BLOCK

// Druck_Temp/R1234ze
(*Wandelt den Druck in die Entsprechende Temperatur um. Die Druck-Temperatur Werte sind in der Nassdampftabelle in den Globalen Variablen hinterlegt.
*)
FUNCTION_BLOCK R1234ze
(*
Versionsverlauf: 
Version		|Autor	|Bemerkung
------------------------------------------------------------------------------------------------------------ 
17.06.00	|Shgb	|erste Freigabe 
17.06.01	|ShgB	|von Integer auf Real geändert	 
17.08.00	|LeaF	|Freigabe

*)
VAR_INPUT
	f_ND:REAL;//Druck für Verdampfungstemperatur
	f_HD:REAL;//Druck für Kondensationstemperatur
END_VAR
VAR_OUTPUT
	f_VerdTemp:REAL;//Verdampfungstemperatur
	f_KondTemp:REAL;//Kondensationstemperatur
END_VAR
VAR
END_VAR

//Niederdruck
	f_VerdTemp:=Nassdampftabelle.R1234ze[REAL_TO_INT(f_ND*100)+100]/10.0;
	
//Hochdruck
	f_KondTemp:=Nassdampftabelle.R1234ze[REAL_TO_INT(f_HD*100)+100]/10.0;

END_FUNCTION_BLOCK

// Druck_Temp/R134a
(*Wandelt den Druck in die Entsprechende Temperatur um. Die Druck-Temperatur Werte sind in der Nassdampftabelle in den Globalen Variablen hinterlegt.
*)
FUNCTION_BLOCK R134a
(*
Versionsverlauf: 
Version		|Autor	|Bemerkung
------------------------------------------------------------------------------------------------------------ 
17.06.00	|Shgb	|erste Freigabe 
17.06.01	|ShgB	|von Integer auf Real geändert	 
17.08.00	|LeaF	|Freigabe

*)
VAR_INPUT
	f_ND:REAL;//Druck für Verdampfungstemperatur
	f_HD:REAL;//Druck für Kondensationstemperatur
END_VAR
VAR_OUTPUT
	f_VerdTemp:REAL;//Verdampfungstemperatur
	f_KondTemp:REAL;//Kondensationstemperatur
END_VAR
VAR
END_VAR

//Niederdruck
	f_VerdTemp:=Nassdampftabelle.R134a[REAL_TO_INT(f_ND*100)+100]/10.0;
	
//Hochdruck
	f_KondTemp:=Nassdampftabelle.R134a[REAL_TO_INT(f_HD*100)+100]/10.0;

END_FUNCTION_BLOCK

// Druck_Temp/R407c
(*Wandelt den Druck in die Entsprechende Temperatur um. Die Druck-Temperatur Werte sind in der Nassdampftabelle in den Globalen Variablen hinterlegt.
*)
FUNCTION_BLOCK R407c
(*
Versionsverlauf: 
Version		|Autor	|Bemerkung
------------------------------------------------------------------------------------------------------------ 
17.06.00	|Shgb	|erste Freigabe 
17.06.01	|ShgB	|von Integer auf Real geändert	 
17.08.00	|LeaF	|Freigabe

*)
VAR_INPUT
	f_ND:REAL;//Druck für Verdampfungstemperatur
	f_HD:REAL;//Druck für Kondensationstemperatur
END_VAR
VAR_OUTPUT
	f_VerdTemp:REAL;//Verdampfungstemperatur
	f_KondTemp:REAL;//Kondensationstemperatur
END_VAR
VAR
END_VAR

//Niederdruck
	f_VerdTemp:=Nassdampftabelle.R407cDew[REAL_TO_INT(f_ND*100)+100]/10.0;
	
//Hochdruck
	f_KondTemp:=Nassdampftabelle.R407cBubble[REAL_TO_INT(f_HD*100)+100]/10.0;

END_FUNCTION_BLOCK

// Druck_Temp/R410a
(*Wandelt den Druck in die Entsprechende Temperatur um. Die Druck-Temperatur Werte sind in der Nassdampftabelle in den Globalen Variablen hinterlegt.
*)
FUNCTION_BLOCK R410a
(*
Versionsverlauf: 
Version		|Autor	|Bemerkung
------------------------------------------------------------------------------------------------------------ 
17.06.00	|Shgb	|erste Freigabe 
17.06.01	|ShgB	|von Integer auf Real geändert	 
17.08.00	|LeaF	|Freigabe

*)
VAR_INPUT
	f_ND:REAL;//Druck für Verdampfungstemperatur
	f_HD:REAL;//Druck für Kondensationstemperatur
END_VAR
VAR_OUTPUT
	f_VerdTemp:REAL;//Verdampfungstemperatur
	f_KondTemp:REAL;//Kondensationstemperatur
END_VAR
VAR
END_VAR

//Niederdruck
	f_VerdTemp:=Nassdampftabelle.R410a[REAL_TO_INT(f_ND*100)+100]/10.0;
	
//Hochdruck
	f_KondTemp:=Nassdampftabelle.R410a[REAL_TO_INT(f_HD*100)+100]/10.0;

END_FUNCTION_BLOCK

// Handschaltungen/HS_Bool
(*Handschaltung für BOOL. 0=> Aus, 1=> Ein und 2=> Automatik.
*)
FUNCTION_BLOCK HS_Bool
(*
Versionsverlauf: 
Version		|Autor	|Bemerkung
------------------------------------------------------------------------------------------------------------ 
17.06.00	|Shgb	|erste Freigabe   
17.08.00	|LeaF	|Freigabe

*)
VAR_INPUT
	x_Ein:BOOL;//Eingang
END_VAR
VAR_INPUT PERSISTENT
	i_Modus:INT;//Modusvorgabe
END_VAR
VAR_OUTPUT
	x_Aus:BOOL;//Ausgang
END_VAR
VAR
END_VAR
VAR CONSTANT
	Ein:INT:=1;
	Aus:INT:=0;
	Auto:INT:=2;
END_VAR

CASE i_Modus OF
	Ein:
		x_Aus:=TRUE;
	Aus:
		x_Aus:=FALSE;
	Auto:
		x_Aus:=x_Ein;
ELSE
	x_Aus:=FALSE;
END_CASE;

END_FUNCTION_BLOCK

// Handschaltungen/HS_Int
(*Handschaltung für INT. 1=> Manuell und 2=> Automatik.
*)
FUNCTION_BLOCK HS_Int
(*
Versionsverlauf: 
Version		|Autor	|Bemerkung
------------------------------------------------------------------------------------------------------------ 
17.06.00	|Shgb	|erste Freigabe   
17.08.00	|LeaF	|Freigabe

*)
VAR_INPUT
	i_Ein:INT;//Eingang
END_VAR
VAR_INPUT PERSISTENT
	i_Manu:INT;//Manuelle Sollstellung
	i_Modus:INT;//Modusvorgabe
END_VAR
VAR_OUTPUT
	i_Aus:INT;//Ausgang
END_VAR
VAR
END_VAR
VAR CONSTANT
	Ein:INT:=1;
	Aus:INT:=0;
	Auto:INT:=2;
END_VAR

CASE i_Modus OF
	Ein:
		i_Aus:=i_Manu;
	Auto:
		i_Aus:=i_Ein;
ELSE
	i_Aus:=0;
END_CASE;

END_FUNCTION_BLOCK

// Handschaltungen/HS_Real
(*Handschaltung für REAL. 1=> Manuell und 2=> Automatik.
*)
FUNCTION_BLOCK HS_Real
(*
Versionsverlauf: 
Version		|Autor	|Bemerkung
------------------------------------------------------------------------------------------------------------ 
17.06.00	|Shgb	|erste Freigabe   
17.08.00	|LeaF	|Freigabe

*)
VAR_INPUT
	f_Ein:REAL;//Eingang
END_VAR
VAR_INPUT PERSISTENT
	f_Manu:REAL;//Manuelle Sollstellung
	i_Modus:INT;//Modusvorgabe
END_VAR
VAR_OUTPUT
	f_Aus:real;//Ausgang
END_VAR
VAR
END_VAR
VAR CONSTANT
	Ein:INT:=1;
	Aus:INT:=0;
	Auto:INT:=2;
END_VAR

CASE i_Modus OF
	Ein:
		f_Aus:=f_Manu;
	Auto:
		f_Aus:=f_Ein;
ELSE
	f_Aus:=0;
END_CASE;

END_FUNCTION_BLOCK

// Heizen_Kuehlen/FG_Heizen
(* Mit der Tagesschaltuhr wird der Tag_Nacht Sollwert bestimmt. Schaltuhr Ein = Nachtbetrieb. Der Funktionsblock wird mit dem Eingang x_Akt aktiviert.
 Unterschreitet die Aussentemperatur und die gemittelte AT den einstellbaren Sollwert
 in der fix eingestellten Zeit von 5 Minuten, schaltet der Einschaltbefehl bis die beiden Temperatur Werte
 der eingestellten Sollwert wieder überschreiten. 
 *)
FUNCTION_BLOCK FG_Heizen
(*
Versionsverlauf: 
Version		|Autor	|Bemerkung
------------------------------------------------------------------------------------------------------------ 
17.07.00	|KuzR	|erste Freigabe  
17.08.00	|LeaF	|Freigabe

*)
VAR_INPUT 
	x_Nacht:BOOL;//Ein=Nacht, Aus=Tag
	f_AT:REAL;//Aussentemperatur
	f_RT_AT:REAL;//Berechnete Aussentemperatur
END_VAR
VAR_INPUT PERSISTENT
	x_Akt_FB:BOOL := TRUE;//Aktivierung FB
	f_SW_Tag:REAL := 20;//Sollwert Tag
	f_SW_Nacht:REAL := 16;//Sollwert Nacht
END_VAR
VAR_OUTPUT
	x_EB:BOOL;//Einschaltbefehl
END_VAR
VAR
	f_Aus_SW_Tag_Nacht:REAL;
	Timer:TON;
	MUX_B: MUX_B;
	x_FG_Tag:BOOL;
	x_FG_Nacht:BOOL;
END_VAR

//Nachtakivierung
	x_FG_Nacht:=x_Akt_FB AND x_Nacht;
	
//Tagaktivierung	
	x_FG_Tag:=x_Akt_FB AND NOT x_Nacht;
	
//Tag/Nacht Umschaltung
	MUX_B(
	f_Ein_1:=f_SW_Tag , 
	f_Ein_2:=f_SW_Nacht , 
	x_Ein_1:=x_FG_Tag , 
	x_Ein_2:=x_FG_Nacht , 
	f_Aus=>f_Aus_SW_Tag_Nacht );
	
//Timer Restzeit für Abfrage AT und SW
	Timer(pt:=T#5M);
	
//Temperaturen Abfrage Tag_Nacht und Timer einschalten
	Timer.IN:= x_Akt_FB AND  f_AT < f_Aus_SW_Tag_Nacht AND f_RT_AT < f_Aus_SW_Tag_Nacht;

//Einschaltbefehl 	
	x_EB:=Timer.Q;

END_FUNCTION_BLOCK

// Heizen_Kuehlen/FG_Kuehlen
(* Mit der Tagesschaltuhr wird der Tag_Nacht Sollwert bestimmt. Schaltuhr Ein = Nachtbetrieb. Der Funktionsblock wird mit dem Eingang x_Akt aktiviert.
 Überschreitet die Aussentemperatur und die gemittelte AT den einstellbaren Sollwert
 in der fix eingestellten Zeit von 5 Min und der Eingang x_Absch_Hz_Kue war länger nicht angezogen, schaltet der Einschaltbefehl bis die beiden Temperatur Werte
 der eingestellten Sollwert wieder unterschreiten. 
 *)
FUNCTION_BLOCK FG_Kuehlen
(*
Versionsverlauf: 
Version		|Autor	|Bemerkung
------------------------------------------------------------------------------------------------------------ 
17.07.00	|KuzR	|erste Freigabe  
17.08.00	|LeaF	|Freigabe

*)
VAR_INPUT 
	x_Nacht: BOOL;//Ein=Nacht, Aus=Tag
	f_AT:REAL;//Aussentemperatur
	f_RT_AT:REAL;//Berechnete Aussentemperatur
END_VAR
VAR_INPUT PERSISTENT
	x_Akt_FB:BOOL := TRUE;//Aktivierung FB
	f_SW_Tag:REAL := 10;//Sollwert Tag
	f_SW_Nacht:REAL := 10;//Sollwert Nacht
	x_Absch_HZ_Kue:BOOL;//Abschaltung HZ und Kühlen
END_VAR
VAR_OUTPUT
	x_EB:BOOL;//Einschaltbefehl
END_VAR
VAR
	f_Aus_SW_Tag_Nacht:REAL;
	Timer:TON;
	MUX_B: MUX_B;
	x_FG_Tag:BOOL;//Freigabe Tag
	x_FG_Nacht:BOOL;//Freigabe Nacht
END_VAR

//Nachtakivierung
	x_FG_Nacht:=x_Akt_FB AND x_Nacht;
	
//Tagaktivierung	
	x_FG_Tag:=x_Akt_FB AND NOT x_Nacht;
	
//Tag/Nacht Umschaltung
	MUX_B(
	f_Ein_1:=f_SW_Tag , 
	f_Ein_2:=f_SW_Nacht , 
	x_Ein_1:=x_FG_Tag , 
	x_Ein_2:=x_FG_Nacht , 
	f_Aus=>f_Aus_SW_Tag_Nacht );	
		
//Timer Restzeit für Abfrage AT und SW
	Timer(pt:=T#5M);	

//Temperaturen Abfrage Tag_Nacht und Timer einschalten
	Timer.IN:= x_Akt_FB AND  f_AT > f_Aus_SW_Tag_Nacht AND f_RT_AT > f_Aus_SW_Tag_Nacht AND NOT x_Absch_HZ_Kue;

//Einschaltbefehl 	
	x_EB:=Timer.Q;

END_FUNCTION_BLOCK

// Heizen_Kuehlen/GR_2
//Kühlkurve, mit 2 AT-Punkten wird ein Tag, bzw. Nachtsollwert berechnet. Referenpunkt T01 muss grösser sein Als T02
//Umschaltbar Tag/Nacht Aktivierung. Sollwert Max und Min Begrenzung. 
FUNCTION_BLOCK GR_2
(*
Versionsverlauf: 
Version		|Autor	|Bemerkung
------------------------------------------------------------------------------------------------------------ 
17.06.00	|KuzR	|erste Freigabe  
17.08.00	|LeaF	|Freigabe

*)
VAR_INPUT
	f_AT:REAL;//Aussentempertur
	x_Akt_Nacht:BOOL;//Nachtakivierung	
END_VAR
VAR_INPUT PERSISTENT
	f_RefPunkt_TO1:REAL;//Referenzpunkt T01 AT
	f_SW_W1_Tag:REAL;//Sollwertpunkt 1 Tag
	f_SW_W1_Nacht:REAL;//Sollwertpunkt 1 Nacht
	f_RefPunkt_TO2:REAL;//Referenzpunkt T02 AT
	f_SW_W2_Tag:REAL;//Sollwertpunkt 2 Tag
	f_SW_W2_Nacht:REAL;//Sollwertpunkt 1 Nacht
	f_SW_Max:REAL;//Sollwert Max.
	f_SW_Min:REAL;//Sollwert Min.
	f_GUI_Zoom:REAL;//Zoomfaktor für das Vergrössern der Grafik
	i_GUI_VersatzX:INT;//Versatz der Grafik in X Richtung (Verdampfung)
	i_GUI_VersatzY:INT;//Versatz der Grafik in Y Richtung (Kondensation)
END_VAR
VAR_OUTPUT
	f_SW_Ber:REAL;//Ausgang Sollwert
END_VAR
	
VAR
	Converter2Punkt: Converter2Punkt;
END_VAR
VAR//Grafik
	f_GUI_RefPunkt_TO1:REAL;//Referenzpunkt T01 AT
	f_GUI_SW_W1_Tag:REAL;//Sollwertpunkt 1 Tag
	f_GUI_SW_W1_Nacht:REAL;//Sollwertpunkt 1 Nacht
	f_GUI_RefPunkt_TO2:REAL;//Referenzpunkt T02 AT
	f_GUI_SW_W2_Tag:REAL;//Sollwertpunkt 2 Tag
	f_GUI_SW_W2_Nacht:REAL;//Sollwertpunkt 1 Nacht
	f_GUI_SW_Max:REAL;//Sollwert Max.
	f_GUI_SW_Min:REAL;//Sollwert Min.
END_VAR

//T01 muss Höher sein als T02
//Aussentemperatur T2-T1, Tag
//Aussentemperatur < T1 oder Aussentemperatur > T2 für Min/Max Begrenzung
	IF NOT x_Akt_Nacht AND  f_RefPunkt_TO2 <= f_AT AND f_RefPunkt_TO1 > f_AT OR NOT x_Akt_Nacht AND f_AT < f_RefPunkt_TO1 OR NOT x_Akt_Nacht AND f_AT > f_RefPunkt_TO2  THEN 
		Converter2Punkt(
	f_Ein:=f_AT , 
	f_Ein_Min:=f_RefPunkt_TO1 , 
	f_Ein_Max:=f_RefPunkt_TO2 , 
	f_Aus_Min:=f_SW_W1_Tag , 
	f_Aus_Max:=f_SW_W2_Tag , 
	f_Aus=>f_SW_Ber );
	END_IF
	
//Aussentemperatur T2-T1, Nacht
//Aussentemperatur < T1 oder Aussentemperatur > T2 für Min/Max Begrenzung
	IF  x_Akt_Nacht AND  
		f_RefPunkt_TO2 <= f_AT AND 
		f_RefPunkt_TO1 > f_AT OR  x_Akt_Nacht AND f_AT < f_RefPunkt_TO1 OR x_Akt_Nacht AND f_AT < f_RefPunkt_TO1 OR  x_Akt_Nacht AND f_AT > f_RefPunkt_TO2  THEN 
		Converter2Punkt(
	f_Ein:=f_AT , 
	f_Ein_Min:=f_RefPunkt_TO1 , 
	f_Ein_Max:=f_RefPunkt_TO2 , 
	f_Aus_Min:=f_SW_W1_Nacht , 
	f_Aus_Max:=f_SW_W2_Nacht , 
	f_Aus=>f_SW_Ber );
	END_IF
	
//Min/Max Begrenzung 
	f_SW_Ber := LIMIT(f_SW_Min,f_SW_Ber, f_SW_Max);

//Grafik für Visu
	f_GUI_RefPunkt_TO1:=f_RefPunkt_TO1 * f_GUI_Zoom + i_GUI_VersatzX;
	f_GUI_SW_W1_Tag:=f_SW_W1_Tag * f_GUI_Zoom + i_GUI_VersatzY * -1;
	f_GUI_SW_W1_Nacht:=f_SW_W1_Nacht * f_GUI_Zoom + i_GUI_VersatzY * -1;
	f_GUI_RefPunkt_TO2:=f_RefPunkt_TO2 * f_GUI_Zoom + i_GUI_VersatzX;
	f_GUI_SW_W2_Tag:=f_SW_W2_Tag * f_GUI_Zoom + i_GUI_VersatzY * -1;
	f_GUI_SW_W2_Nacht:=f_SW_W2_Nacht * f_GUI_Zoom + i_GUI_VersatzY * -1;
	f_GUI_SW_Max:= f_SW_Max * f_GUI_Zoom + i_GUI_VersatzY * -1;
	f_GUI_SW_Min:= f_SW_Min * f_GUI_Zoom + i_GUI_VersatzY * -1;

END_FUNCTION_BLOCK

// Heizen_Kuehlen/GR_4_mit_RE
(* Heizkurve mit Raumeinfluss vergleicht Aussentemperatur zwischen den Sollwerten. Referenzpunkt T01 muss die kleinste Temperatur-,bzw. T04 die grösste Temperatur sein.
 Anhand von vier AT Punkten wird der Tag-, bzw. Nachtsollwert berechnet.
 Umschaltbar Tag/Nacht Aktivierung. Sollwert mit  Max und Min Begrenzung. Maximale negative Korrektur (i_MaxKorrNeg) muss zwingend als negativen Wert eingegeben werden und Maximale positive  Korrektur als positiven Wert.
*)
FUNCTION_BLOCK GR_4_mit_RE
(*
Versionsverlauf: 
Version		|Autor	|Bemerkung
------------------------------------------------------------------------------------------------------------ 
17.06.00	|KuzR	|erste Freigabe  
17.08.00	|LeaF	|Freigabe

*)
VAR_INPUT
	f_AT:REAL; //Aussentemperatur
	x_Akt_Nacht:BOOL;	// Nachtakivierung
	f_MT_Raum:REAL; // Raumtemperatur
END_VAR
VAR_INPUT PERSISTENT	
	f_RefPunkt_TO1:REAL; // Referenzpunkt T01 AT
	f_SW_W1_Tag:REAL; // Sollwertpunkt 1 Tag
	f_SW_W1_Nacht:REAL; // Sollwertpunkt 1 Nacht
	f_RefPunkt_TO2:REAL; // Referenzpunkt T02 AT
	f_SW_W2_Tag:REAL; // Sollwertpunkt 2 Tag
	f_SW_W2_Nacht:REAL; // Sollwertpunkt 2 Nacht
	f_RefPunkt_TO3:REAL; // Referenzpunkt T03 AT
	f_SW_W3_Tag:REAL; // Sollwertpunkt 3 Tag
	f_SW_W3_Nacht:REAL; // Sollwertpunkt 3 Nacht
	f_RefPunkt_TO4:REAL; // Referenzpunkt T04 AT
	f_SW_W4_Tag:REAL; // Sollwertpunkt 4 Tag
	f_SW_W4_Nacht:REAL; // Sollwertpunkt 4 Nacht
	f_SW_Max:REAL; // Sollwert Max.
	f_SW_Min:REAL; //Sollwert Min.
	f_KorrFaktor:REAL;  // Korrekturfaktor
	i_MaxKorrPos:INT; // Max. Pos. Korrektur(muss positiver Wert sein)
	i_MaxKorrNeg:INT; // Max. Neg. Korrektur(muss negativer Wert sein)
	f_SW_Raum:REAL;	// Sollwert Raum
	f_GUI_Zoom:REAL;//Zoomfaktor für das Vergrössern der Grafik
	i_GUI_VersatzX:INT;//Versatz der Grafik in X Richtung (Verdampfung)
	i_GUI_VersatzY:INT;//Versatz der Grafik in Y Richtung (Kondensation)
END_VAR
VAR_OUTPUT
	f_SW_Ber:REAL; // Sollwert Berechnung
	f_SW_Korr:REAL; // Korrigierte Sollwertberechnung
END_VAR
VAR
	f_Diff:REAL;
	f_Diff_faktor:REAL;
	Converter2Punkt: Converter2Punkt;
END_VAR
VAR//Grafik
	f_GUI_RefPunkt_TO1:REAL;//Referenzpunkt T01 AT
	f_GUI_SW_W1_Tag:REAL;//Sollwertpunkt 1 Tag
	f_GUI_SW_W1_Nacht:REAL;//Sollwertpunkt 1 Nacht
	f_GUI_RefPunkt_TO2:REAL;//Referenzpunkt T02 AT
	f_GUI_SW_W2_Tag:REAL;//Sollwertpunkt 2 Tag
	f_GUI_SW_W2_Nacht:REAL;//Sollwertpunkt 2 Nacht
	f_GUI_RefPunkt_TO3:REAL;//Referenzpunkt T03 AT
	f_GUI_SW_W3_Tag:REAL;//Sollwertpunkt 3 Tag
	f_GUI_SW_W3_Nacht:REAL;//Sollwertpunkt 3 Nacht
	f_GUI_RefPunkt_TO4:REAL;//Referenzpunkt T04 AT
	f_GUI_SW_W4_Tag:REAL;//Sollwertpunkt 4 Tag
	f_GUI_SW_W4_Nacht:REAL;//Sollwertpunkt 4 Nacht
	f_GUI_SW_Max:REAL;//Sollwert Max.
	f_GUI_SW_Min:REAL;//Sollwert Min.
END_VAR

//Aussentemperatur T4-T3, Tag
//Aussentemperatur > T4, für Max Sollwert Berechnung
	IF NOT x_Akt_Nacht AND f_RefPunkt_TO4 > f_AT AND f_RefPunkt_TO3 <= f_AT OR NOT x_Akt_Nacht AND f_AT >= f_RefPunkt_TO4 THEN
		Converter2Punkt( 
	f_Ein:=f_AT , 
	f_Ein_Min:=f_RefPunkt_TO3 , 
	f_Ein_Max:=f_RefPunkt_TO4 , 
	f_Aus_Min:=f_SW_W3_Tag , 
	f_Aus_Max:=f_SW_W4_Tag , 
	f_Aus=>f_SW_Ber );
	END_IF
//Aussentemperatur T4-T3, Nacht
//Aussentemperatur > T4, für Max Sollwert Berechnung
	IF x_Akt_Nacht AND f_RefPunkt_TO4 > f_AT AND f_RefPunkt_TO3 <= f_AT OR x_Akt_Nacht AND f_AT >= f_RefPunkt_TO4 THEN
		Converter2Punkt(
	f_Ein:=f_AT , 
	f_Ein_Min:=f_RefPunkt_TO3 , 
	f_Ein_Max:=f_RefPunkt_TO4 , 
	f_Aus_Min:=f_SW_W3_Nacht , 
	f_Aus_Max:=f_SW_W4_Nacht , 
	f_Aus=>f_SW_Ber );
	END_IF
//Aussentemperatur T3-T2, Tag
	IF NOT x_Akt_Nacht AND  f_RefPunkt_TO3 > f_AT AND f_RefPunkt_TO2 <= f_AT THEN
		Converter2Punkt(
	f_Ein:=f_AT , 
	f_Ein_Min:=f_RefPunkt_TO2 , 
	f_Ein_Max:=f_RefPunkt_TO3 , 
	f_Aus_Min:=f_SW_W2_Tag , 
	f_Aus_Max:=f_SW_W3_Tag , 
	f_Aus=>f_SW_Ber );
	END_IF
//Aussentemperatur T3-T2, Nacht
	IF x_Akt_Nacht AND  f_RefPunkt_TO3 > f_AT AND f_RefPunkt_TO2 <= f_AT THEN
		Converter2Punkt(
	f_Ein:=f_AT , 
	f_Ein_Min:=f_RefPunkt_TO2 , 
	f_Ein_Max:=f_RefPunkt_TO3 , 
	f_Aus_Min:=f_SW_W2_Nacht , 
	f_Aus_Max:=f_SW_W3_Nacht , 
	f_Aus=>f_SW_Ber );
	END_IF	
//Aussentemperatur T2-T1, Tag
//Aussentemperatur < T1, für Min Sollwert Berechnung
	IF NOT x_Akt_Nacht AND f_RefPunkt_TO2 > f_AT AND f_RefPunkt_TO1 <= f_AT OR NOT x_Akt_Nacht AND f_AT < f_RefPunkt_TO1  THEN
		Converter2Punkt(
	f_Ein:=f_AT , 
	f_Ein_Min:=f_RefPunkt_TO1 , 
	f_Ein_Max:=f_RefPunkt_TO2 , 
	f_Aus_Min:=f_SW_W1_Tag , 
	f_Aus_Max:=f_SW_W2_Tag , 
	f_Aus=>f_SW_Ber );
	END_IF
//Aussentemperatur T2-T1, Nacht
//Aussentemperatur < T1, für Min Sollwert Berechnung
	IF x_Akt_Nacht AND f_RefPunkt_TO2 > f_AT AND f_RefPunkt_TO1 <= f_AT OR x_Akt_Nacht AND f_AT < f_RefPunkt_TO1  THEN
		Converter2Punkt(
	f_Ein:=f_AT , 
	f_Ein_Min:=f_RefPunkt_TO1 , 
	f_Ein_Max:=f_RefPunkt_TO2 , 
	f_Aus_Min:=f_SW_W1_Nacht , 
	f_Aus_Max:=f_SW_W2_Nacht , 
	f_Aus=>f_SW_Ber );
	END_IF

//Korrektur Raumtemperatur
	f_Diff:= f_SW_Raum-f_MT_Raum;
	
//Maximale_Minimale Korrektur
	IF f_Diff > i_MaxKorrPos THEN
		f_Diff:=i_MaxKorrPos;
	END_IF
	IF f_Diff < i_MaxKorrNeg THEN
		f_Diff:=i_MaxKorrNeg;
	END_IF
	
	f_Diff_faktor:=f_Diff*f_KorrFaktor;
	
//Begrenzung für positive und negative Begerenzung
	IF f_Diff_faktor > i_MaxKorrPos THEN
		f_Diff_faktor:=i_MaxKorrPos;
	END_IF
	IF f_Diff_faktor < i_MaxKorrNeg THEN
		f_Diff_faktor:=i_MaxKorrNeg;
	END_IF
	
//Korrrigierter Sollwert	
	f_SW_Korr:=f_SW_Ber + f_Diff_faktor ;

//Max Begrenzung 	
	IF f_SW_Korr >= f_SW_Max THEN
		f_SW_Korr:=f_SW_Max; 
	END_IF	
//Min Begrenzung 
	IF f_SW_Korr < f_SW_Min THEN
		f_SW_Korr:=f_SW_Min;
	END_IF


//Grafik für Visu
	f_GUI_RefPunkt_TO1:=f_RefPunkt_TO1 * f_GUI_Zoom + i_GUI_VersatzX;
	f_GUI_SW_W1_Tag:=f_SW_W1_Tag * f_GUI_Zoom + i_GUI_VersatzY * -1;
	f_GUI_SW_W1_Nacht:=f_SW_W1_Nacht * f_GUI_Zoom + i_GUI_VersatzY * -1;
	f_GUI_RefPunkt_TO2:=f_RefPunkt_TO2 * f_GUI_Zoom + i_GUI_VersatzX;
	f_GUI_SW_W2_Tag:=f_SW_W2_Tag * f_GUI_Zoom + i_GUI_VersatzY * -1;
	f_GUI_SW_W2_Nacht:=f_SW_W2_Nacht * f_GUI_Zoom + i_GUI_VersatzY * -1;
	f_GUI_RefPunkt_TO3:=f_RefPunkt_TO3 * f_GUI_Zoom + i_GUI_VersatzX;
	f_GUI_SW_W3_Tag:=f_SW_W3_Tag * f_GUI_Zoom + i_GUI_VersatzY * -1;
	f_GUI_SW_W3_Nacht:=f_SW_W3_Nacht * f_GUI_Zoom + i_GUI_VersatzY * -1;
	f_GUI_RefPunkt_TO4:=f_RefPunkt_TO4 * f_GUI_Zoom + i_GUI_VersatzX;
	f_GUI_SW_W4_Tag:=f_SW_W4_Tag * f_GUI_Zoom + i_GUI_VersatzY * -1;
	f_GUI_SW_W4_Nacht:=f_SW_W4_Nacht * f_GUI_Zoom + i_GUI_VersatzY * -1;
	f_GUI_SW_Max:= f_SW_Max * f_GUI_Zoom + i_GUI_VersatzY * -1;
	f_GUI_SW_Min:= f_SW_Min * f_GUI_Zoom + i_GUI_VersatzY * -1;

END_FUNCTION_BLOCK

// Heizen_Kuehlen/GR_4_ohne_RE
(* Heizkurve ohne Raumeinfluss vergleicht Aussentemperatur zwischen den Sollwerten. Referenzpunkt T01 muss die kleinste Temperatur-,bzw. T04 die grösste Temperatur sein.
 Anhand von vier AT Punkten wird der Tag-, bzw. Nachtsollwert berechnet.
 Umschaltbar Tag/Nacht Aktivierung. Sollwert MAX und MIN Begrenzung.
*)
FUNCTION_BLOCK GR_4_ohne_RE
(*
Versionsverlauf: 
Version		|Autor	|Bemerkung
------------------------------------------------------------------------------------------------------------ 
17.06.00	|KuzR	|erste Freigabe  
17.08.00	|LeaF	|Freigabe

*)
VAR_INPUT
	f_AT:REAL; //Aussentemperatur
	x_Akt_Nacht:BOOL;//Nachtakivierung
END_VAR
VAR_INPUT PERSISTENT
	f_RefPunkt_TO1:REAL;//Referenzpunkt T01 AT
	f_SW_W1_Tag:REAL;//Sollwertpunkt 1 Tag
	f_SW_W1_Nacht:REAL;//Sollwertpunkt 1 Nacht
	f_RefPunkt_TO2:REAL;//Referenzpunkt T02 AT
	f_SW_W2_Tag:REAL;//Sollwertpunkt 2 Tag
	f_SW_W2_Nacht:REAL;//Sollwertpunkt 2 Nacht
	f_RefPunkt_TO3:REAL;//Referenzpunkt T03 AT
	f_SW_W3_Tag:REAL;//Sollwertpunkt 3 Tag
	f_SW_W3_Nacht:REAL;//Sollwertpunkt 3 Nacht
	f_RefPunkt_TO4:REAL;//Referenzpunkt T04 AT
	f_SW_W4_Tag:REAL;//Sollwertpunkt 4 Tag
	f_SW_W4_Nacht:REAL;//Sollwertpunkt 4 Nacht
	f_SW_Max:REAL;//Sollwert Max.
	f_SW_Min:REAL;//Sollwert Min.
	f_GUI_Zoom:REAL;//Zoomfaktor für das Vergrössern der Grafik
	i_GUI_VersatzX:INT;//Versatz der Grafik in X Richtung (Verdampfung)
	i_GUI_VersatzY:INT;//Versatz der Grafik in Y Richtung (Kondensation)
END_VAR
VAR_OUTPUT
	f_SW_Ber:REAL;//Sollwert Berechnung
END_VAR
VAR
	Converter2Punkt: Converter2Punkt;
END_VAR
VAR//Grafik
	f_GUI_RefPunkt_TO1:REAL;//Referenzpunkt T01 AT
	f_GUI_SW_W1_Tag:REAL;//Sollwertpunkt 1 Tag
	f_GUI_SW_W1_Nacht:REAL;//Sollwertpunkt 1 Nacht
	f_GUI_RefPunkt_TO2:REAL;//Referenzpunkt T02 AT
	f_GUI_SW_W2_Tag:REAL;//Sollwertpunkt 2 Tag
	f_GUI_SW_W2_Nacht:REAL;//Sollwertpunkt 2 Nacht
	f_GUI_RefPunkt_TO3:REAL;//Referenzpunkt T03 AT
	f_GUI_SW_W3_Tag:REAL;//Sollwertpunkt 3 Tag
	f_GUI_SW_W3_Nacht:REAL;//Sollwertpunkt 3 Nacht
	f_GUI_RefPunkt_TO4:REAL;//Referenzpunkt T04 AT
	f_GUI_SW_W4_Tag:REAL;//Sollwertpunkt 4 Tag
	f_GUI_SW_W4_Nacht:REAL;//Sollwertpunkt 4 Nacht
	f_GUI_SW_Max:REAL;//Sollwert Max.
	f_GUI_SW_Min:REAL;//Sollwert Min.
END_VAR

//Aussentemperatur T4-T3, Tag
//Aussentemperatur > T4, für Max Sollwert Berechnung
	IF NOT x_Akt_Nacht AND f_RefPunkt_TO4 > f_AT AND f_RefPunkt_TO3 <= f_AT OR NOT x_Akt_Nacht AND f_AT >= f_RefPunkt_TO4 THEN
		Converter2Punkt( 
	f_Ein:=f_AT , 
	f_Ein_Min:=f_RefPunkt_TO3 , 
	f_Ein_Max:=f_RefPunkt_TO4 , 
	f_Aus_Min:=f_SW_W3_Tag , 
	f_Aus_Max:=f_SW_W4_Tag , 
	f_Aus=>f_SW_Ber );
	END_IF
//Aussentemperatur T4-T3, Nacht
//Aussentemperatur > T4, für Max Sollwert Berechnung
	IF x_Akt_Nacht AND f_RefPunkt_TO4 > f_AT AND f_RefPunkt_TO3 <= f_AT OR x_Akt_Nacht AND f_AT >= f_RefPunkt_TO4 THEN
		Converter2Punkt(
	f_Ein:=f_AT , 
	f_Ein_Min:=f_RefPunkt_TO3 , 
	f_Ein_Max:=f_RefPunkt_TO4 , 
	f_Aus_Min:=f_SW_W3_Nacht , 
	f_Aus_Max:=f_SW_W4_Nacht , 
	f_Aus=>f_SW_Ber );
	END_IF
//Aussentemperatur T3-T2, Tag
	IF NOT x_Akt_Nacht AND  f_RefPunkt_TO3 > f_AT AND f_RefPunkt_TO2 <= f_AT THEN
		Converter2Punkt(
	f_Ein:=f_AT , 
	f_Ein_Min:=f_RefPunkt_TO2 , 
	f_Ein_Max:=f_RefPunkt_TO3 , 
	f_Aus_Min:=f_SW_W2_Tag , 
	f_Aus_Max:=f_SW_W3_Tag , 
	f_Aus=>f_SW_Ber );
	END_IF
//Aussentemperatur T3-T2, Nacht
	IF x_Akt_Nacht AND  f_RefPunkt_TO3 > f_AT AND f_RefPunkt_TO2 <= f_AT THEN
		Converter2Punkt(
	f_Ein:=f_AT , 
	f_Ein_Min:=f_RefPunkt_TO2 , 
	f_Ein_Max:=f_RefPunkt_TO3 , 
	f_Aus_Min:=f_SW_W2_Nacht , 
	f_Aus_Max:=f_SW_W3_Nacht , 
	f_Aus=>f_SW_Ber );
	END_IF	
//Aussentemperatur T2-T1, Tag
//Aussentemperatur < T1, für Min Sollwert Berechnung
	IF NOT x_Akt_Nacht AND f_RefPunkt_TO2 > f_AT AND f_RefPunkt_TO1 <= f_AT OR NOT x_Akt_Nacht AND f_AT < f_RefPunkt_TO1  THEN
		Converter2Punkt(
	f_Ein:=f_AT , 
	f_Ein_Min:=f_RefPunkt_TO1 , 
	f_Ein_Max:=f_RefPunkt_TO2 , 
	f_Aus_Min:=f_SW_W1_Tag , 
	f_Aus_Max:=f_SW_W2_Tag , 
	f_Aus=>f_SW_Ber );
	END_IF
//Aussentemperatur T2-T1, Nacht
//Aussentemperatur < T1, für Min Sollwert Berechnung
	IF x_Akt_Nacht AND f_RefPunkt_TO2 > f_AT AND f_RefPunkt_TO1 <= f_AT OR x_Akt_Nacht AND f_AT < f_RefPunkt_TO1  THEN
		Converter2Punkt(
	f_Ein:=f_AT , 
	f_Ein_Min:=f_RefPunkt_TO1 , 
	f_Ein_Max:=f_RefPunkt_TO2 , 
	f_Aus_Min:=f_SW_W1_Nacht , 
	f_Aus_Max:=f_SW_W2_Nacht , 
	f_Aus=>f_SW_Ber );
	END_IF

//Min/Max Begrenzung 	
	f_SW_Ber := LIMIT(f_SW_Min,f_SW_Ber, f_SW_Max);

	
//Grafik für Visu
	f_GUI_RefPunkt_TO1:=f_RefPunkt_TO1 * f_GUI_Zoom + i_GUI_VersatzX;
	f_GUI_SW_W1_Tag:=f_SW_W1_Tag * f_GUI_Zoom + i_GUI_VersatzY * -1;
	f_GUI_SW_W1_Nacht:=f_SW_W1_Nacht * f_GUI_Zoom + i_GUI_VersatzY * -1;
	f_GUI_RefPunkt_TO2:=f_RefPunkt_TO2 * f_GUI_Zoom + i_GUI_VersatzX;
	f_GUI_SW_W2_Tag:=f_SW_W2_Tag * f_GUI_Zoom + i_GUI_VersatzY * -1;
	f_GUI_SW_W2_Nacht:=f_SW_W2_Nacht * f_GUI_Zoom + i_GUI_VersatzY * -1;
	f_GUI_RefPunkt_TO3:=f_RefPunkt_TO3 * f_GUI_Zoom + i_GUI_VersatzX;
	f_GUI_SW_W3_Tag:=f_SW_W3_Tag * f_GUI_Zoom + i_GUI_VersatzY * -1;
	f_GUI_SW_W3_Nacht:=f_SW_W3_Nacht * f_GUI_Zoom + i_GUI_VersatzY * -1;
	f_GUI_RefPunkt_TO4:=f_RefPunkt_TO4 * f_GUI_Zoom + i_GUI_VersatzX;
	f_GUI_SW_W4_Tag:=f_SW_W4_Tag * f_GUI_Zoom + i_GUI_VersatzY * -1;
	f_GUI_SW_W4_Nacht:=f_SW_W4_Nacht * f_GUI_Zoom + i_GUI_VersatzY * -1;
	f_GUI_SW_Max:= f_SW_Max * f_GUI_Zoom + i_GUI_VersatzY * -1;
	f_GUI_SW_Min:= f_SW_Min * f_GUI_Zoom + i_GUI_VersatzY * -1;

END_FUNCTION_BLOCK

// Heizen_Kuehlen/REG2_HEIZEN
(*2 Punkt Regler Heizen
Für Direkt, x_Akt auf true, schaltet der Ausgang auf true. Ist der eingegebene Sollwert addiert mit dem Einschaltpunkt(zB -2) grösser oder gleich der Messtemperatur,
schaltet der digitale Ausgang auf true. Ist der Sollwert addiert mit dem Ausschaltpunkt kleiner oder gleich dem Messwert, schaltet der digitale Ausganf auf false.
*)
FUNCTION_BLOCK REG2_HEIZEN
(*
Versionsverlauf: 
Version		|Autor	|Bemerkung
------------------------------------------------------------------------------------------------------------ 
17.06.00	|KuzR	|erste Freigabe  
17.08.00	|LeaF	|Freigabe

*)
VAR_INPUT
	f_MT:REAL;//Eingang Messwert
END_VAR
VAR_INPUT PERSISTENT
	f_SW:REAL;//Eingang Sollwert
	f_Einschaltpunkt:REAL;//Eingang Einschaltpunkt
	f_Ausschaltpunkt:REAL;//Eingang Ausschaltpunkt
	x_Akt:BOOL;//Direkt-Indirekt Aktivierung
END_VAR
VAR_OUTPUT
	x_Aus:BOOL;//Digitaler Ausgang
END_VAR
VAR
END_VAR

//Direkt- Indirekt Schaltung
	IF   NOT x_Akt THEN 
		x_Aus:=FALSE;
//Einschalten
	ELSIF  f_MT <= f_SW + f_Einschaltpunkt THEN
		x_Aus:= TRUE;
//Ausschalten	
	ELSIF	f_MT  >= f_SW + f_Ausschaltpunkt THEN
		x_Aus:= FALSE;
	END_IF

END_FUNCTION_BLOCK

// Heizen_Kuehlen/REG2_KUEHLEN
(*2 Punkt Regler Kühlen
Für Direkt, x_Akt auf true, schaltet der Ausgang auf true. Ist der eingegebene Sollwert addiert mit dem Einschaltpunkt(zB -2) kleiner oder gleich der Messtemperatur,
schaltet der digitale Ausgang auf true. Ist der Sollwert addiert mit dem Ausschaltpunkt grösser oder gleich dem Messwert, schaltet der digitale Ausganf auf false.
*)
FUNCTION_BLOCK REG2_KUEHLEN
(*
Versionsverlauf: 
Version		|Autor	|Bemerkung
------------------------------------------------------------------------------------------------------------ 
17.06.00	|KuzR	|erste Freigabe  
17.08.00	|LeaF	|Freigabe

*)
VAR_INPUT
	f_MT:REAL;//Eingang Messwert
END_VAR
VAR_INPUT PERSISTENT
	f_SW:REAL;//Eingang Sollwert
	f_Einschaltpunkt:REAL;//Eingang Einschaltpunkt
	f_Ausschaltpunkt:REAL;//Eingang Ausschaltpunkt
	x_Akt:BOOL;//Direkt-Indirekt Aktivierung
END_VAR
VAR_OUTPUT
	x_Aus:BOOL;//Digitaler Ausgang
END_VAR
VAR
END_VAR

//Direkt- Indirekt Schaltung
	IF   NOT x_Akt THEN 
		x_Aus:=FALSE;	
//Einschalten
	ELSIF  f_MT >= f_SW + f_Einschaltpunkt THEN
		x_Aus:= TRUE;	
//Ausschalten	
	ELSIF	f_MT  <= f_SW + f_Ausschaltpunkt THEN
		x_Aus:= FALSE;	
	END_IF

END_FUNCTION_BLOCK

// Heizen_Kuehlen/RT_AT_48
(*Berechnet die gemittelte Aussentemperatur. Die Datensätze für die Mittelwertberechnung ist auf 48 Datensätze ausgelegt.
x_start für die Initialisierung der Aussentemperatur. Mit t_time kann die Zeit bestimmt werden, wann einen Wert ins Array geschrieben werden kann.
*)
FUNCTION_BLOCK RT_AT_48
(*
Versionsverlauf: 
Version		|Autor	|Bemerkung
------------------------------------------------------------------------------------------------------------ 
17.07.00	|KuzR	|erste Freigabe  
17.08.00	|LeaF	|Freigabe

*)
VAR_INPUT
	x_start: BOOL;//Start für die  Initialisierung
	f_AT:REAL;//Eingang Aussentemperatur
END_VAR
VAR_INPUT PERSISTENT	
	t_time:timestruct;//Zeiteingabe 1h oder 24h
END_VAR
VAR_OUTPUT
	f_AT_RT: REAL;//Ausgang gemittelt
END_VAR
VAR 
	i_Ind: INT;
	f_Summe:REAL;
	timer:ton;
	daten:ARRAY [1..i_Datensaetze] OF REAL;
	Timestruct_to_Time:Timestruct_to_Time;	
	x_Flanke: BOOL;
END_VAR
VAR CONSTANT
	i_Datensaetze:INT:=48;
END_VAR

//Für Aussentemperatur Initialisierung muss x_start gedrückt werden
	 IF x_start  THEN
//Grösse des Array für den Mittelwert bestimmen
		 FOR i_Ind:= 1 TO I_DATENSAETZE DO
			 daten[i_Ind]:= f_AT;
		 END_FOR
	 END_IF
	x_start:=FALSE;
//Timestruct to Time
	timestruct_to_time(t_Ein:=t_time);
//Timer läuft immer
	Timer(IN := NOT Timer.Q, PT :=timestruct_to_time.t_Aus/48 );

	IF Timer.Q THEN
    f_Summe := 0;
//die neuen Temperaturwerte werden ins Array geschrieben
    FOR i_Ind := I_DATENSAETZE TO 2 BY -1  DO
        Daten[i_Ind] := Daten[i_Ind - 1];
        f_Summe := f_Summe + Daten[i_Ind];
    END_FOR
//Rechentemperatur berechnen
    Daten[1] := f_AT;
    f_Summe := f_Summe + f_AT;
    f_AT_RT:=f_summe / I_DATENSAETZE;
	END_IF

END_FUNCTION_BLOCK

// Initialisierung/Globale_Zeit
FUNCTION_BLOCK Globale_Zeit
(*
Versionsverlauf: 
Version		|Autor	|Bemerkung
------------------------------------------------------------------------------------------------------------ 
17.06.00	|KuzR	|erste Freigabe 
17.06.01	|ShgB	|Date and Time ergänzt 
17.08.00	|LeaF	|Freigabe

*)
VAR_INPUT Persistent
	tzi_ZeitZone:ST_TimeZoneInformation :=WEST_EUROPE_TZI;
	x_SetTime: BOOL;
	t_NewTime:timestruct;
END_VAR
VAR_OUTPUT		 
END_VAR
VAR
	  fbgetSystemTime:getsystemtime;
  	  fileTime:T_FILETIME;
	  
      eTzID:E_TimeZoneID := eTimeZoneID_Unknown;
      fbToLocal:FB_FileTimeToTzSpecificLocalTime;
	  tzInfo:ST_TimeZoneInformation;
	  NT_SetLocalTime:NT_SetLocalTime;
END_VAR

//CPU Zeit
	fbgetSystemTime	(timeLoDW=>fileTime.dwLowDateTime, timeHiDW=>fileTime.dwHighDateTime );
	
//Zeitumrechnung
	fbToLocal( in := filetime , tzInfo := tzi_ZeitZone );
	
//Globale Variable, Aktuelle Uhrzeit
	Globale_Uhr.systemtimestruct := FILETIME_TO_systemtime( fbToLocal.out  );
	Globale_Uhr.systemDateAndTime:= FILETIME_TO_DT(fbToLocal.out);
	
//Zeit setzen
	NT_SetLocalTime(TIMESTR:= t_NewTime, START:= x_SetTime );

END_FUNCTION_BLOCK

// Math/Average
(*Gibt den Durchschnitt der angeschlossenen Werten aus.
*)
FUNCTION_BLOCK Average
(*
Versionsverlauf: 
Version		|Autor	|Bemerkung
------------------------------------------------------------------------------------------------------------ 
17.06.00	|Shgb	|erste Freigabe  
17.08.00	|LeaF	|Freigabe

*)
VAR_INPUT
	f_Ein1 :REAL:=0.00001;//Wert 1
	f_Ein2 :REAL:=0.00001;//Wert 2
	f_Ein3 :REAL:=0.00001;//Wert 3
	f_Ein4 :REAL:=0.00001;//Wert 4
	f_Ein5 :REAL:=0.00001;//Wert 5
	f_Ein6 :REAL:=0.00001;//Wert 6
	f_Ein7 :REAL:=0.00001;//Wert 7
	f_Ein8 :REAL:=0.00001;//Wert 8
END_VAR
VAR_OUTPUT
	f_Aus:REAL;//Durchschnitt
END_VAR
VAR
	i_Arraypos:INT;
	af_Array: ARRAY [1..8] OF REAL;
	COUNT: COUNT;
END_VAR

// Werte in Array platzieren
	af_Array[1]:=f_Ein1;
	af_Array[2]:=f_Ein2;
	af_Array[3]:=f_Ein3;
	af_Array[4]:=f_Ein4;
	af_Array[5]:=f_Ein5;
	af_Array[6]:=f_Ein6;
	af_Array[7]:=f_Ein7;
	af_Array[8]:=f_Ein8;
	
//Zurücksetzen
	f_Aus:=0;
	
//Anzahl Eingänge zählen
	COUNT(
	x_Ein_1:= f_Ein1<>0.00001, //0.00001 bedeutet nicht aktiv
	x_Ein_2:= f_Ein2<>0.00001, 
	x_Ein_3:= f_Ein3<>0.00001, 
	x_Ein_4:= f_Ein4<>0.00001, 
	x_Ein_5:= f_Ein5<>0.00001, 
	x_Ein_6:= f_Ein6<>0.00001, 
	x_Ein_7:= f_Ein7<>0.00001, 
	x_Ein_8:= f_Ein8<>0.00001);
	
//Summe bilden
	FOR i_Arraypos:=1 TO count.i_Aus DO
		f_Aus:=f_Aus+af_Array[i_Arraypos];
	END_FOR
	
//Durchschnitt berechnen
	IF count.i_Aus >0 THEN
		f_Aus:=f_Aus/count.i_Aus;
	END_IF

END_FUNCTION_BLOCK

// Math/Filter
(*Berechnet die gefilterte Aussentemperatur. x_start für die Initialisierung der Aussentemperatur. Mit t_time kann die Zeit bestimmt werden, wann einen Wert ins Array geschrieben werden kann.
*)
FUNCTION_BLOCK Filter
(*
Versionsverlauf:
Version		|Autor	|Bemerkung
------------------------------------------------------------------------------------------------------------ 
17.07.00	|KuzR	|erste Freigabe  
17.08.00	|LeaF	|Freigabe

*)
VAR_INPUT
	x_start: BOOL;//Start für die  Initialisierung
	f_AT:REAL;//Eingang Aussentemperatur
END_VAR
VAR_INPUT PERSISTENT	
	t_time:timestruct := (wHour := 1);//Takt, wenn ein AT Wert geschrieben wird
END_VAR
VAR_OUTPUT
	f_Aus: REAL;//Ausgang gefiltert
END_VAR
VAR 
	i_Ind: INT;
	f_Summe:REAL;
	timer:ton;
	daten:ARRAY [1..i_Datensaetze] OF REAL;
	Timestruct_to_Time:Timestruct_to_Time;	
	x_Flanke: BOOL;
END_VAR
VAR CONSTANT
	i_Datensaetze:INT:=48;
END_VAR

//Für Aussentemperatur Initialisierung muss x_start gedrückt werden
	 IF x_start  THEN
//Grösse des Array für den Mittelwert bestimmen
		 FOR i_Ind:= 1 TO I_DATENSAETZE DO
			 daten[i_Ind]:= f_AT;
		 END_FOR
	 END_IF
		x_start:=FALSE;
//Timestruct to Time
	timestruct_to_time(t_Ein:=t_time);
//Timer läuft immer
	Timer(IN := NOT Timer.Q, PT :=timestruct_to_time.t_Aus );

	IF Timer.Q THEN
    f_Summe := 0;
//die neuen Temperaturwerte werden ins Array geschrieben
    FOR i_Ind := I_DATENSAETZE TO 2 BY -1  DO
        Daten[i_Ind] := Daten[i_Ind - 1];
        f_Summe := f_Summe + Daten[i_Ind];
    END_FOR
//Rechentemperatur berechnen
    Daten[1] := f_AT;
    f_Summe := f_Summe + f_AT;
    f_Aus:=f_summe / I_DATENSAETZE;
	END_IF

END_FUNCTION_BLOCK

// Math/Minimun
(*Gibt den kleinsten der angeschlossenen Werten aus.
*)
FUNCTION_BLOCK Minimun
(*
Versionsverlauf: 
Version		|Autor	|Bemerkung
------------------------------------------------------------------------------------------------------------ 
17.06.00	|Shgb	|erste Freigabe 
17.06.01	|ShgB	|von Integer auf Real geändert	 
17.08.00	|LeaF	|Freigabe

*)
VAR_INPUT
	f_Ein1 :REAL:=0.00001;//Wert 1
	f_Ein2 :REAL:=0.00001;//Wert 2
	f_Ein3 :REAL:=0.00001;//Wert 3
	f_Ein4 :REAL:=0.00001;//Wert 4
	f_Ein5 :REAL:=0.00001;//Wert 5
	f_Ein6 :REAL:=0.00001;//Wert 6
	f_Ein7 :REAL:=0.00001;//Wert 7
	f_Ein8 :REAL:=0.00001;//Wert 8
END_VAR
VAR_OUTPUT
	f_Aus:REAL;//Kleinste Wert
END_VAR
VAR
	i_Arraypos:INT;
	af_Array: ARRAY [1..8] OF REAL;
END_VAR

// Werte in Array platzieren
	af_Array[1]:=f_Ein1;
	af_Array[2]:=f_Ein2;
	af_Array[3]:=f_Ein3;
	af_Array[4]:=f_Ein4;
	af_Array[5]:=f_Ein5;
	af_Array[6]:=f_Ein6;
	af_Array[7]:=f_Ein7;
	af_Array[8]:=f_Ein8;
		
//Zahlen die grösser als 0 sind
	f_Aus := af_Array[1];	
	
//Auswertung der kleinsten Zahl
	FOR i_Arraypos:=2 TO 8 DO
		IF af_Array[i_Arraypos] <= f_Aus AND af_Array[i_Arraypos] <> 0.00001 THEN
			f_Aus := af_Array[i_Arraypos];
		END_IF
	END_FOR

END_FUNCTION_BLOCK

// Math/Range
(*Wertet aus ob sich der Eingang im angegebenen Bereich befindet. Wert in Grenzen => Ausgang False Wert ausserhalb => Ausgang True
*)
FUNCTION_BLOCK Range
(*
Versionsverlauf: 
Version		|Autor	|Bemerkung
------------------------------------------------------------------------------------------------------------ 
17.06.00	|Shgb	|erste Freigabe  
17.08.00	|LeaF	|Freigabe

*)
VAR_INPUT
	f_Ein:REAL;//Eingang
	f_Min:REAL;//Eingangsbereich Minimum
	f_Max:REAL;//Eingangsbereich Maximum
END_VAR
VAR_OUTPUT
	x_Aus:BOOL;//Ausgang
END_VAR
VAR
END_VAR

x_Aus:= not (f_Ein<=f_Max and f_Ein>=f_Min);

END_FUNCTION_BLOCK

// Math/Timestruct_Kleiner_Gleich_Timestruct
(*Vergleicht zweit Timestructvariablen. Wenn die erste kleiner oder gleich ist wird der Ausgang TRUE andernfalls bleit der Ausgang FALSE
*)
FUNCTION_BLOCK Timestruct_Kleiner_Gleich_Timestruct
(*
Versionsverlauf: 
Version		|Autor	|Bemerkung
------------------------------------------------------------------------------------------------------------ 
17.08.00	|ShgB	|erste Freigabe 

*)
VAR_INPUT
	t_Ein1:TIMESTRUCT;//Referenztimestruct
	t_Ein2:Timestruct;//Vergleichstimestruct
END_VAR
VAR_OUTPUT
	x_Aus:BOOL;//True wenn Vergleichtimestruct kleiner Referenztimestruct ist
END_VAR
VAR
END_VAR

x_Aus:=FALSE;
IF t_Ein1.wDay < t_Ein2.wDay THEN
	x_Aus:=TRUE;
ELSIF t_Ein1.wDay = t_Ein2.wDay THEN
	IF t_Ein1.wHour < t_Ein2.wHour THEN
		x_Aus:=TRUE;
	ELSIF t_Ein1.wHour = t_Ein2.wHour THEN
		IF t_Ein1.wMinute < t_Ein2.wMinute THEN
			x_Aus:=TRUE;
		ELSIF t_Ein1.wMinute = t_Ein2.wMinute THEN
			IF t_Ein1.wSecond < t_Ein2.wSecond THEN
				x_Aus:=TRUE;
			ELSIF t_Ein1.wSecond = t_Ein2.wSecond THEN
				IF t_Ein1.wMilliseconds <= t_Ein2.wMilliseconds THEN
					x_Aus:=TRUE;
				END_IF
			END_IF
		END_IF
	END_IF
END_IF

END_FUNCTION_BLOCK

// Memory/Logger
(*Loggt die angegebenen Datenpunkte im entsprechenden Takt und speichert diese für den angegebenen Zeitraum ab.
*)
FUNCTION_BLOCK Logger
(*
Versionsverlauf: 
Version		|Autor	|Bemerkung
------------------------------------------------------------------------------------------------------------ 
17.07.00	|Shgb	|erste Freigabe  
17.08.00	|LeaF	|Freigabe

*)
VAR_INPUT PERSISTENT
	s_Dir:STRING(255):='C:\TwinCAT\Logger';//Dateipfad für Logdateien
	s_Filename:STRING(255):='Log';//Name der Datei. Wird mit JJJJ_MM_DD ergänzt
	t_Takt:Timestruct := (wSecond := 5);//Takt der Aufzeichnung
	i_Speicherdauer:INT:=14;//Anzahl Tage die gespeichert werden
END_VAR
VAR_INPUT
	x_Ein:BOOL;//Öffent eine Datei und Loggt die Datenpunkte
	x_Record:BOOL;//Datenpunkte werden unabhängig des Taktes geloggts_Titel1:STRING(255);//Titel 1-32 des Datenpunktes
	s_Titel1:STRING(255);//Datenpunkttitel für Kopfzeile
	f_Data1: REAL;//Datenpunkt 1-32
	i_Dezimalstelle1:INT;//Anzahl Dezimalstellen 1-32
	s_Titel2:STRING(255);
	f_Data2: REAL;
	i_Dezimalstelle2:INT;
	s_Titel3:STRING(255);
	f_Data3: REAL;
	i_Dezimalstelle3:INT;
	s_Titel4:STRING(255);
	f_Data4: REAL;
	i_Dezimalstelle4:INT;
	s_Titel5:STRING(255);
	f_Data5: REAL;
	i_Dezimalstelle5:INT;
	s_Titel6:STRING(255);
	f_Data6: REAL;
	i_Dezimalstelle6:INT;
	s_Titel7:STRING(255);
	f_Data7: REAL;
	i_Dezimalstelle7:INT;
	s_Titel8:STRING(255);
	f_Data8: REAL;
	i_Dezimalstelle8:INT;
	s_Titel9:STRING(255);
	f_Data9: REAL;
	i_Dezimalstelle9:INT;
	s_Titel10:STRING(255);
	f_Data10: REAL;
	i_Dezimalstelle10:INT;
	s_Titel11:STRING(255);
	f_Data11: REAL;
	i_Dezimalstelle11:INT;
	s_Titel12:STRING(255);
	f_Data12: REAL;
	i_Dezimalstelle12:INT;
	s_Titel13:STRING(255);
	f_Data13: REAL;
	i_Dezimalstelle13:INT;
	s_Titel14:STRING(255);
	f_Data14: REAL;
	i_Dezimalstelle14:INT;
	s_Titel15:STRING(255);
	f_Data15: REAL;
	i_Dezimalstelle15:INT;
	s_Titel16:STRING(255);
	f_Data16: REAL;
	i_Dezimalstelle16:INT;
	s_Titel17:STRING(255);
	f_Data17: REAL;
	i_Dezimalstelle17:INT;
	s_Titel18:STRING(255);
	f_Data18: REAL;
	i_Dezimalstelle18:INT;
	s_Titel19:STRING(255);
	f_Data19: REAL;
	i_Dezimalstelle19:INT;
	s_Titel20:STRING(255);
	f_Data20: REAL;
	i_Dezimalstelle20:INT;
	s_Titel21:STRING(255);
	f_Data21: REAL;
	i_Dezimalstelle21:INT;
	s_Titel22:STRING(255);
	f_Data22: REAL;
	i_Dezimalstelle22:INT;
	s_Titel23:STRING(255);
	f_Data23: REAL;
	i_Dezimalstelle23:INT;
	s_Titel24:STRING(255);
	f_Data24: REAL;
	i_Dezimalstelle24:INT;
	s_Titel25:STRING(255);
	f_Data25: REAL;
	i_Dezimalstelle25:INT;
	s_Titel26:STRING(255);
	f_Data26: REAL;
	i_Dezimalstelle26:INT;
	s_Titel27:STRING(255);
	f_Data27: REAL;
	i_Dezimalstelle27:INT;
	s_Titel28:STRING(255);
	f_Data28: REAL;
	i_Dezimalstelle28:INT;
	s_Titel29:STRING(255);
	f_Data29: REAL;
	i_Dezimalstelle29:INT;
	s_Titel30:STRING(255);
	f_Data30: REAL;
	i_Dezimalstelle30:INT;
	s_Titel31:STRING(255);
	f_Data31: REAL;
	i_Dezimalstelle31:INT;
	s_Titel32:STRING(255);
	f_Data32: REAL;
	i_Dezimalstelle32:INT;
END_VAR
VAR_OUTPUT
	x_FileOpen:BOOL;//Datei geöffnet
	x_AL_Open:BOOL;//Fehler beim Öffnen der Datei
	x_AL_Write:BOOL;//Fehler beim schreiben der Datenpunkte
	x_AL_Close:BOOL;//Fehler beim Schliessen der Datei
	x_AL_Delete:BOOL;//Fehler beim Löschen der Datei (Datei nicht existent)
END_VAR
VAR
	as_Array:ARRAY[0..33] OF STRING;
	af_Array:ARRAY [1..32] OF REAL;
	ai_Array:ARRAY [1..32] OF INT;
	i_Schrittkette:INT;
	i_Arraypos:INT;
	s_File:STRING;
	s_DelFile:STRING;
	s_temp: STRING;
	s_Data:STRING;
	s_DT: STRING(255);
	f_temp: REAL;
	i_Dezimalzeichen: INT;
	i_LastFile:UINT;
	Timer: TON;
	t_Speicherdauer: TIMESTRUCT;
	Timestruct_to_Time:Timestruct_to_Time;
	FB_CreateDir:FB_CreateDir;
	FB_FileOpen: FB_FileOpen;
	FB_FilePuts: FB_FilePuts;
	FB_FileClose: FB_FileClose;
	FB_FileDelete: FB_FileDelete;
END_VAR
VAR CONSTANT
	I_INIT: INT := 0;
	I_CREATE_DIR: INT := 1;
	I_WAIT_DIR: INT := 2;
	I_FILE_OPEN: INT := 3;
	I_WAIT_OPEN: INT := 4;
	I_FILE_Header: INT := 5;
	I_WAIT_Header: INT := 6;
	I_FILE_WRITE: INT := 7;
	I_END_WRITE: INT := 8;
	I_WAIT_WRITE: INT := 9;
	I_FILE_CLOSE: INT := 10;
	I_WAIT_CLOSE: INT := 11;
END_VAR

//Datenerfassung
	as_Array[0]:='Datum;Zeit;';
	as_Array[1]:=concat(s_Titel1,';');
	as_Array[2]:=concat(s_Titel2,';');
	as_Array[3]:=concat(s_Titel3,';');
	as_Array[4]:=concat(s_Titel4,';');
	as_Array[5]:=concat(s_Titel5,';');
	as_Array[6]:=concat(s_Titel6,';');
	as_Array[7]:=concat(s_Titel7,';');
	as_Array[8]:=concat(s_Titel8,';');
	as_Array[9]:=concat(s_Titel9,';');
	as_Array[10]:=concat(s_Titel10,';');
	as_Array[11]:=concat(s_Titel11,';');
	as_Array[12]:=concat(s_Titel12,';');
	as_Array[13]:=concat(s_Titel13,';');
	as_Array[14]:=concat(s_Titel14,';');
	as_Array[15]:=concat(s_Titel15,';');
	as_Array[16]:=concat(s_Titel16,';');
	as_Array[17]:=concat(s_Titel17,';');
	as_Array[18]:=concat(s_Titel18,';');
	as_Array[19]:=concat(s_Titel19,';');
	as_Array[20]:=concat(s_Titel20,';');
	as_Array[21]:=concat(s_Titel21,';');
	as_Array[22]:=concat(s_Titel22,';');
	as_Array[23]:=concat(s_Titel23,';');
	as_Array[24]:=concat(s_Titel24,';');
	as_Array[25]:=concat(s_Titel25,';');
	as_Array[26]:=concat(s_Titel26,';');
	as_Array[27]:=concat(s_Titel27,';');
	as_Array[28]:=concat(s_Titel28,';');
	as_Array[29]:=concat(s_Titel29,';');
	as_Array[30]:=concat(s_Titel30,';');
	as_Array[31]:=concat(s_Titel31,';');
	as_Array[32]:=concat(s_Titel32,';');
	as_Array[33]:='$N';
	
	af_Array[1]:=f_Data1;
	af_Array[2]:=f_Data2;
	af_Array[3]:=f_Data3;
	af_Array[4]:=f_Data4;
	af_Array[5]:=f_Data5;
	af_Array[6]:=f_Data6;
	af_Array[7]:=f_Data7;
	af_Array[8]:=f_Data8;
	af_Array[9]:=f_Data9;
	af_Array[10]:=f_Data10;
	af_Array[11]:=f_Data11;
	af_Array[12]:=f_Data12;
	af_Array[13]:=f_Data13;
	af_Array[14]:=f_Data14;
	af_Array[15]:=f_Data15;
	af_Array[16]:=f_Data16;
	af_Array[17]:=f_Data17;
	af_Array[18]:=f_Data18;
	af_Array[19]:=f_Data19;
	af_Array[20]:=f_Data20;
	af_Array[21]:=f_Data21;
	af_Array[22]:=f_Data22;
	af_Array[23]:=f_Data23;
	af_Array[24]:=f_Data24;
	af_Array[25]:=f_Data25;
	af_Array[26]:=f_Data26;
	af_Array[27]:=f_Data27;
	af_Array[28]:=f_Data28;
	af_Array[29]:=f_Data29;
	af_Array[30]:=f_Data30;
	af_Array[31]:=f_Data31;
	af_Array[32]:=f_Data32;
	
	ai_Array[1]:=i_Dezimalstelle1;
	ai_Array[2]:=i_Dezimalstelle2;
	ai_Array[3]:=i_Dezimalstelle3;
	ai_Array[4]:=i_Dezimalstelle4;
	ai_Array[5]:=i_Dezimalstelle5;
	ai_Array[6]:=i_Dezimalstelle6;
	ai_Array[7]:=i_Dezimalstelle7;
	ai_Array[8]:=i_Dezimalstelle8;
	ai_Array[9]:=i_Dezimalstelle9;
	ai_Array[10]:=i_Dezimalstelle10;
	ai_Array[11]:=i_Dezimalstelle11;
	ai_Array[12]:=i_Dezimalstelle12;
	ai_Array[13]:=i_Dezimalstelle13;
	ai_Array[14]:=i_Dezimalstelle14;
	ai_Array[15]:=i_Dezimalstelle15;
	ai_Array[16]:=i_Dezimalstelle16;
	ai_Array[17]:=i_Dezimalstelle17;
	ai_Array[18]:=i_Dezimalstelle18;
	ai_Array[19]:=i_Dezimalstelle19;
	ai_Array[20]:=i_Dezimalstelle20;
	ai_Array[21]:=i_Dezimalstelle21;
	ai_Array[22]:=i_Dezimalstelle22;
	ai_Array[23]:=i_Dezimalstelle23;
	ai_Array[24]:=i_Dezimalstelle24;
	ai_Array[25]:=i_Dezimalstelle25;
	ai_Array[26]:=i_Dezimalstelle26;
	ai_Array[27]:=i_Dezimalstelle27;
	ai_Array[28]:=i_Dezimalstelle28;
	ai_Array[29]:=i_Dezimalstelle29;
	ai_Array[30]:=i_Dezimalstelle30;
	ai_Array[31]:=i_Dezimalstelle31;
	ai_Array[32]:=i_Dezimalstelle32;
	

//Dateiname erstellen
	s_File:=CONCAT(STR1:=s_Dir, STR2:='\');
	s_File:=CONCAT(STR1:=s_File, STR2:=s_Filename);
	s_File:=CONCAT(STR1:=s_File, STR2:='_');
	s_File:=CONCAT(STR1:=s_File, STR2:=DWORD_TO_STRING(Globale_Uhr.systemtimestruct.wYear));
	s_File:=CONCAT(STR1:=s_File, STR2:='_');
	s_File:=CONCAT(STR1:=s_File, STR2:=DWORD_TO_STRING(Globale_Uhr.systemtimestruct.wMonth));
	s_File:=CONCAT(STR1:=s_File, STR2:='_');
	s_File:=CONCAT(STR1:=s_File, STR2:=DWORD_TO_STRING(Globale_Uhr.systemtimestruct.wDay));
	s_File:=CONCAT(STR1:=s_File, STR2:='.csv');

//Pfad für zu löschende Datei
	t_Speicherdauer:=DT_TO_SYSTEMTIME( Globale_Uhr.systemDateAndTime-i_Speicherdauer*T#1D-T#1D);
				
	s_DelFile:=CONCAT(STR1:=s_Dir, STR2:='\');
	s_DelFile:=CONCAT(STR1:=s_DelFile, STR2:=s_Filename);
	s_DelFile:=CONCAT(STR1:=s_DelFile, STR2:='_');
	s_DelFile:=CONCAT(STR1:=s_DelFile, STR2:=DWORD_TO_STRING(t_Speicherdauer.wYear));
	s_DelFile:=CONCAT(STR1:=s_DelFile, STR2:='_');
	s_DelFile:=CONCAT(STR1:=s_DelFile, STR2:=DWORD_TO_STRING(t_Speicherdauer.wMonth));
	s_DelFile:=CONCAT(STR1:=s_DelFile, STR2:='_');
	s_DelFile:=CONCAT(STR1:=s_DelFile, STR2:=DWORD_TO_STRING(t_Speicherdauer.wDay));
	s_DelFile:=CONCAT(STR1:=s_DelFile, STR2:='.csv');

//Datum und Uhrzeit erstellen
	s_DT:='';
	s_DT:=CONCAT(STR1:=s_DT, STR2:=DWORD_TO_STRING(Globale_Uhr.systemtimestruct.wDay));
	s_DT:=CONCAT(STR1:=s_DT, STR2:='.');
	s_DT:=CONCAT(STR1:=s_DT, STR2:=DWORD_TO_STRING(Globale_Uhr.systemtimestruct.wMonth));
	s_DT:=CONCAT(STR1:=s_DT, STR2:='.');
	s_DT:=CONCAT(STR1:=s_DT, STR2:=DWORD_TO_STRING(Globale_Uhr.systemtimestruct.wYear));
	s_DT:=CONCAT(STR1:=s_DT, STR2:=';');
	s_DT:=CONCAT(STR1:=s_DT, STR2:=DWORD_TO_STRING(Globale_Uhr.systemtimestruct.wHour));
	s_DT:=CONCAT(STR1:=s_DT, STR2:=':');
	s_DT:=CONCAT(STR1:=s_DT, STR2:=DWORD_TO_STRING(Globale_Uhr.systemtimestruct.wMinute));
	s_DT:=CONCAT(STR1:=s_DT, STR2:=':');
	s_DT:=CONCAT(STR1:=s_DT, STR2:=DWORD_TO_STRING(Globale_Uhr.systemtimestruct.wSecond));			

//Timestruct to Time
	Timestruct_to_Time(t_Ein:=t_Takt);
	
//Takt
	Timer(IN:= x_Ein AND NOT Timer.Q, PT:= Timestruct_to_Time.t_Aus);
	
//Case
	CASE i_Schrittkette OF
		I_INIT:
			IF x_Ein THEN
				i_Schrittkette:=I_CREATE_DIR;
			END_IF
		
		I_CREATE_DIR:
			FB_CreateDir.bExecute:=TRUE;
			i_Schrittkette:=I_WAIT_DIR;
	
		I_WAIT_DIR:
			IF NOT FB_CreateDir.bBusy THEN
				i_Schrittkette:=I_FILE_OPEN;
				FB_CreateDir.bExecute:=FALSE;
			END_IF
		
		I_FILE_OPEN:
			FB_FileOpen.sPathName:=s_File;
			FB_FileOpen.bExecute:=TRUE;
			i_Schrittkette:= I_WAIT_OPEN;
			
		I_WAIT_OPEN:
			IF NOT FB_FileOpen.bBusy AND FB_FileOpen.hFile <> 0 AND FB_FileOpen.hFile <> i_LastFile THEN
				IF s_File <> s_temp THEN
					i_Schrittkette:=I_FILE_Header;
					FB_FileDelete.bExecute:=TRUE;
					s_temp:=s_File;
				ELSE
					i_Schrittkette:=I_WAIT_WRITE;
					FB_FileDelete.bExecute:=FALSE;	
				END_IF
				i_Arraypos:=0;
				FB_FileOpen.bExecute:=FALSE;
			END_IF
			IF NOT FB_FileOpen.bBusy AND (FB_FileOpen.hFile = 0 OR FB_FileOpen.hFile = i_LastFile)  THEN
				i_Schrittkette:=I_FILE_OPEN;
				FB_FileOpen.bExecute:=FALSE;
			END_IF
			
		I_FILE_Header:
			FB_FilePuts.sLine:=as_Array[i_Arraypos];
			IF LEN(as_Array[i_Arraypos])>0 THEN 
				FB_FilePuts.bExecute:=TRUE;
			END_IF
			i_Schrittkette:= I_WAIT_Header;
			i_Arraypos:=i_Arraypos+1;
		
		I_WAIT_Header:
			IF NOT FB_FilePuts.bBusy AND i_Arraypos <=33 THEN
				i_Schrittkette:=I_FILE_Header;
				FB_FilePuts.bExecute:=FALSE;
			END_IF
			IF NOT FB_FilePuts.bBusy AND i_Arraypos =34 THEN
				i_Schrittkette:=I_WAIT_WRITE;
				i_Arraypos:=0;
				FB_FilePuts.bExecute:=FALSE;
			END_IF
						
		I_WAIT_WRITE:
			IF NOT FB_FilePuts.bBusy AND i_Arraypos<=33 THEN
				i_Schrittkette:=I_FILE_WRITE;
				FB_FilePuts.bExecute:=FALSE;
			END_IF
			IF NOT FB_FilePuts.bBusy AND i_Arraypos>33 THEN
				i_Schrittkette:=I_END_WRITE;
				i_Arraypos:=0;
				FB_FilePuts.bExecute:=FALSE;
			END_IF
		
		I_FILE_WRITE:
			CASE i_Arraypos OF
				0:
					FB_FilePuts.sLine:=concat(STR1:= s_DT,STR2:=';');
				
				1..32:
					s_Data:='';
					s_Data:=CONCAT(STR1:=s_Data,STR2:=DINT_TO_STRING(TRUNC(af_Array[i_Arraypos])));
					IF ai_Array[i_Arraypos] >0 THEN
						s_Data:=CONCAT(STR1:=s_Data, STR2:='.');
						f_temp:=af_Array[i_Arraypos]-TRUNC(af_Array[i_Arraypos]);
						FOR i_Dezimalzeichen:=1 TO ai_Array[i_Arraypos] DO
							f_temp:=f_temp*10;
						END_FOR
					s_Data:=CONCAT(STR1:=s_Data,STR2:=DINT_TO_STRING(TRUNC(f_temp)));
					END_IF
					s_Data:=CONCAT(STR1:=s_Data, STR2:=';');
					FB_FilePuts.sLine:=s_Data;				
				
				33:
					FB_FilePuts.sLine:='$N';
			END_CASE
			IF LEN(as_Array[i_Arraypos])>0 THEN 
				FB_FilePuts.bExecute:=TRUE;
			END_IF
			i_Schrittkette:= I_WAIT_WRITE;
			i_Arraypos:=i_Arraypos+1;	

		I_END_WRITE:
			IF Timer.Q THEN
				i_Schrittkette:=I_FILE_WRITE;
			END_IF
			
			IF NOT x_Ein OR s_File <> s_temp THEN
				i_Schrittkette:=I_FILE_CLOSE;
			END_IF	
			
		I_FILE_CLOSE:
			FB_FileClose.bExecute:=TRUE;
			i_Schrittkette:= I_WAIT_CLOSE;
			
		I_WAIT_CLOSE:
			IF NOT FB_FileClose.bBusy THEN
				FB_FileClose.bExecute:=FALSE;
				i_LastFile:=FB_FileOpen.hFile;
				i_Schrittkette:=I_INIT;
			END_IF
	END_CASE

//FB Create Dir
	FB_CreateDir(
		sPathName:= s_Dir);
				
//FB File Open
	FB_FileOpen( 
		nMode:= FOPEN_MODEAPPEND OR FOPEN_MODEPLUS,
		bError=> x_AL_Open);
		
//FB File Write
	FB_FilePuts( 
				hFile:= FB_FileOpen.hFile,
				bError=> x_AL_Write);
				
//FB File Close
	FB_FileClose(
				hFile:= FB_FileOpen.hFile,
				bError=> x_AL_Close);
				
//File Open
	x_FileOpen:=i_Schrittkette>=I_WAIT_Header;
	
//FB Delete File
	FB_FileDelete( 
		sPathName:= s_DelFile, 
		bError=> x_AL_Delete);

END_FUNCTION_BLOCK

// Regler/EEV
(*Dieser Funktionsbaustein regelt die Verdampfungstemperatur, mittels EEV, um den Überhitzungssollwert tiefer als die Sauggastemperatur.
Formel: Soll Verdampfung = Sauggastemperatur - Überhitzungssollwert
Die Soll Verdampfung wird zudem noch durch den MOP begrenzt. Ist die Überhitzung länger als 2 Minuten unterhalb von 2K so wird ein Alarm ausgelöst.
*)
FUNCTION_BLOCK EEV
(*
Versionsverlauf: 
Version		|Autor	|Bemerkung
------------------------------------------------------------------------------------------------------------ 
17.06.00	|Shgb	|erste Freigabe 
17.06.01	|ShgB	|von Integer auf Real geändert	
17.06.02	|ShgB	|Von Time auf Timestruct geändert
17.08.00	|LeaF	|Freigabe

*)
VAR_INPUT
	x_Enable:BOOL;//Regelung Freigeben
	f_Verdampfunstemperatur:REAL;//Verdampfungstemperatur
	f_Sauggastemperatur:REAL;//Sauggastemperatur
	x_SW_Reset:BOOL;//Setzt die Standardwerte für den Verdichterty zurück
	f_MOP_Einsatzgrenzen: REAL := 0.00001;//Dynamischer MOP von Einsatzgrenzen
	dut_Verdichtertyp:SW_Einsatzgrenzen:=SW_ALZ.Bitzer_Scroll_R410a;//Verdichtertyp als DUT Angabe Standard Bitzer Scroll 410a
END_VAR
VAR_INPUT PERSISTENT
	f_SollwertUBH:REAL := 6;//Sollwert für die Überhitzung
	f_MOP:REAL;//Maximal Operating Pressure
	f_PFaktor:REAL:=3.0;//P Faktor für Regelung
	f_IFaktor:REAL:=0.05;//I Faktor für Regelung
	f_DFaktor:REAL:=0;//D Faktor für Regelung
	t_Takt:timestruct := (wMilliseconds := 100);//Berechnungstakt des PID Reglers
	f_MinUBH:REAL:=2;//Minimale Überhitzung
	t_AL_EEV:Timestruct := (wMinute := 2);//Zeit bis Alarm ausgelöst wird
END_VAR
VAR_OUTPUT
	f_UBH:REAL;//Berechnete Überhitzung
	f_Regelsignal:REAL;//Regelsignal für das Expansionsventil
	x_Alarm:BOOL;//Überhitzung wurde nicht erreicht/
END_VAR
VAR
	f_SollVerdampfung:REAL;
	PID: PIDRegler;
	UBH_Timer: TON;
	x_TempAlarm: BOOL;
	Timestruct_to_Time: Timestruct_to_Time;
END_VAR

VAR PERSISTENT
	x_Laden: BOOL;//Variable ist beim ersten aufstarten False und lädt somit die eingestellten Daten
END_VAR

//Überhitzung 
	f_UBH:=f_Sauggastemperatur-f_Verdampfunstemperatur;
	
//Soll Verdampfungstemperatur berechnen
	f_SollVerdampfung:=f_Sauggastemperatur-f_SollwertUBH;
	//MOP 
	IF f_SollVerdampfung > f_MOP_Einsatzgrenzen AND f_MOP_Einsatzgrenzen <> 0.00001 THEN
		f_SollVerdampfung:=f_MOP_Einsatzgrenzen;
	END_IF
	
	IF f_SollVerdampfung > f_MOP THEN
		f_SollVerdampfung:=f_MOP;
	END_IF
	
//PID Regelung
	PID(
		x_Enable:= x_Enable and not x_Alarm, 
		x_Invertiert:= FALSE, 
		x_Manuell:= FALSE, 
		f_Sollwert:= f_SollVerdampfung, 
		f_Ist:= f_Verdampfunstemperatur, 
		f_Offset:= 0, 
		f_Min:= 0, 
		f_Max:= 100, 
		f_Manuell:= 0, 
		f_PFaktor:= f_PFaktor, 
		f_IFaktor:= f_IFaktor, 
		f_DFaktor:= f_DFaktor, 
		t_Takt:= t_Takt, 
		f_Regelsignal=> f_Regelsignal);
		
//Überhitzungsschutz < 2K
	IF f_UBH < f_MinUBH THEN
		f_Regelsignal:=f_Regelsignal/2;
	END_IF

//Alarm
	IF Globale_Variablen.x_Quittieren THEN
		x_Alarm:=FALSE;
	END_IF
	
	//Timestruct to Time
	Timestruct_to_Time(t_Ein:= t_AL_EEV);
	
	UBH_Timer(IN:= f_UBH<2.0 AND x_Enable, PT:= Timestruct_to_Time.t_Aus, Q=> x_TempAlarm, ET=> );
	
	IF x_TempAlarm THEN
		x_Alarm:=TRUE;
	END_IF	
	
//Reset Sollwerte
	IF x_SW_Reset OR NOT x_Laden THEN
		f_MOP:=dut_Verdichtertyp.f_SW_EG_MaxVerd-2;
		x_Laden:=TRUE;
	END_IF

END_FUNCTION_BLOCK

// Regler/PIDRegler
(*Der PID Regler rechnet die Differenz zwischen dem Sollwert und dem Istwert aus und multipliziert diese mit dem P Faktor. 
Die I und D Anteile werden bei jedem Takt neu berechnet und auf den P Anteil dazu addiert. 
Je grösser die Faktoren sind, desto schneller und instabiler wirde der Regler.
P Anteil: 
Formel Normal: (Sollwert + Ossfet - Istwert) x P Faktor 
Formel Invertiert: (Istwert - Sollwert - Offset) x P Faktor 
I Anteil: 
Formel: I Anteil + I Faktor x P Anteil 
D Anteil: 
Formel: (P Anteil - P Anteil (vom letzten Takt)) x D Faktor
Regelsignal: P + I + D Anteil
*)
FUNCTION_BLOCK PIDRegler
(*
Versionsverlauf: 
Version		|Autor	|Bemerkung
------------------------------------------------------------------------------------------------------------ 
17.06.00	|Shgb	|erste Freigabe 
17.06.01	|ShgB	|von Integer auf Real geändert	
17.06.02	|ShgB	|Von Time auf Timestruct geändert
17.07.00	|ShgB	|Offset und Invertierung geändert.
17.08.00	|LeaF	|Freigabe	

*)
VAR_INPUT
	x_Enable:BOOL;//Freigabe des Reglers
	f_Ist:REAL;//Istwert
END_VAR
VAR_INPUT PERSISTENT
	x_Invertiert:BOOL;//Bei Kühlfunktionen aktiv
	x_Manuell:BOOL;//Manuelles Regelsignal aktivieren
	f_Sollwert:REAL;//Sollwertvorgabe
	f_Offset:REAL;//Offset
	f_Min:REAL;//Minimales Regelsignal
	f_Max:REAL;//Maximales Regelsignal
	f_Manuell:REAL;//Manuelles Regelsignal
	f_PFaktor:REAL;//Proportionalfaktor
	f_IFaktor:REAL;//Integralfaktor
	f_DFaktor:REAL;//Differenzialfaktor
	t_Takt:timestruct;//Regelungstakt
END_VAR
VAR_OUTPUT
	f_Regelsignal:REAL;//Regelsignal
END_VAR
VAR
	f_IAnteil,f_ISpeicher,f_DAnteil:REAL;
	f_PAnteil,f_DSpeicher:REAL;
	P_Anteil: PRegler;
	Timer: TON;
	x_Takt:BOOL;
	Timestruct_to_Time: Timestruct_to_Time;
END_VAR

//P Anteil	
	P_Anteil(
		x_Enable:= x_Enable, 
		x_Invertiert:= x_Invertiert, 
		x_Manuell:= FALSE, 
		f_Sollwert:= f_Sollwert, 
		f_Ist:= f_Ist, 
		f_Offset:= f_Offset, 
		f_Min:= -f_Max, 
		f_Max:= f_Max, 
		f_Manuell:= 0, 
		f_PFaktor:= f_PFaktor, 
		f_Regelsignal=> f_PAnteil);
		
//TImestruct to Time
	Timestruct_to_Time(t_Ein:=t_Takt);	

//Takt
	Timer(IN:= x_Enable AND NOT x_Takt, PT:= Timestruct_to_Time.t_Aus, Q=> x_Takt, ET=> );
	
//I Anteil
	IF x_Takt AND f_Regelsignal<f_Max AND f_Regelsignal>f_Min THEN
		f_ISpeicher:=f_ISpeicher+f_IFaktor*f_PAnteil;
	END_IF

//D Anteil
	IF x_Takt THEN
		f_DAnteil:=(f_PAnteil-f_DSpeicher)*f_DFaktor;
		f_DSpeicher:=f_PAnteil;
	END_IF

//Reset Speicher
	IF NOT x_Enable THEN
		f_ISpeicher:=0.0;
		f_DSpeicher:=0.0;
	END_IF

//Grenzen einhalten	
	f_Regelsignal := LIMIT(f_Min,f_ISpeicher+f_DAnteil+f_PAnteil, f_Max);

//Manuell	
	IF x_Manuell THEN
		f_Regelsignal:=f_Manuell;
	END_IF

END_FUNCTION_BLOCK

// Regler/PRegler
(*Der P Regler rechnet die Differenz zwischen dem Sollwert und dem Istwert aus und multipliziert diese mit dem P Faktor. Je grösser der Faktor ist, desto schneller und instabiler wirde der Regler.
Formel Normal: (Sollwert + Ossfet - Istwert) x P Faktor 
Formel Invertiert: (Istwert - Sollwert - Offset) x P Faktor 
*)
FUNCTION_BLOCK PRegler
(*
Versionsverlauf: 
Version		|Autor	|Bemerkung
------------------------------------------------------------------------------------------------------------ 
17.06.00	|Shgb	|erste Freigabe 
17.06.01	|ShgB	|von Integer auf Real geändert	
17.07.00	|ShgB	|Offset und Invertierung geändert.	
17.08.00	|LeaF	|Freigabe

*)
VAR_INPUT
	x_Enable:BOOL;//Freigabe des Reglers
	f_Ist:REAL;//Istwert
END_VAR
VAR_INPUT PERSISTENT
	x_Invertiert:BOOL;//Bei Kühlfunktionen aktiv
	x_Manuell:BOOL;//Manuelles Regelsignal aktivieren
	f_Sollwert:REAL;//Sollwertvorgabe
	f_Offset:REAL;//Offset
	f_Min:REAL;//Minimales Regelsignal
	f_Max:REAL;//Maximales Regelsignal
	f_Manuell:REAL;//Manuelles Regelsignal
	f_PFaktor:REAL;//Proportionalfaktor
	t_Takt:timestruct;//Regelungstakt
END_VAR
VAR_OUTPUT
	f_Regelsignal:REAL;//Regelsignal
END_VAR
VAR
END_VAR

IF x_Enable THEN//Wenn Ein wird berechnet	
	IF x_Manuell THEN//Wenn Manuell wird der Manuelle Wert auf den Ausgang geschrieben
		f_Regelsignal:=LIMIT(f_Min,f_Manuell,f_Max);
	ELSE//Sonst wird die Berechnung durchgeführt
		IF x_Invertiert THEN//Formel für Berechnung (Istwert - Sollwert - Offset) x P Faktor 
			f_Regelsignal:=LIMIT(f_Min,
							(f_Ist-f_Sollwert-f_Offset)*f_PFaktor,
							f_Max);
		ELSE//(Sollwert + Ossfet - Istwert) x P Faktor 
			f_Regelsignal:=LIMIT(f_Min,
							(f_Sollwert+f_Offset-f_Ist)*f_PFaktor,
							f_Max);
		END_IF
		
	END_IF
ELSE//Sonst wird Regelsignal auf 0 geschrieben
	f_Regelsignal:=0.0;
END_IF

END_FUNCTION_BLOCK

// Regler/PIRegler
(*Der PI Regler rechnet die Differenz zwischen dem Sollwert und dem Istwert aus und multipliziert diese mit dem P Faktor. 
Zudem rechnet er bei jedem Takt den I Anteil aus und addiert diesen auf mit dem P Anteil. Je grösser die Faktoren sind, desto schneller und instabiler wirde der Regler.
P Anteil:
Formel Normal: (Sollwert + Ossfet - Istwert) x P Faktor 
Formel Invertiert: (Istwert - Sollwert - Offset) x P Faktor 
I Anteil:
Formel: I Anteil + I Faktor x P Anteil
Regelsignal: P + I Anteil
*)
FUNCTION_BLOCK PIRegler
(*
Versionsverlauf: 
Version		|Autor	|Bemerkung
------------------------------------------------------------------------------------------------------------ 
17.06.00	|Shgb	|erste Freigabe 
17.06.01	|ShgB	|von Integer auf Real geändert	
17.06.02	|ShgB	|Von Time auf Timestruct geändert
17.07.00	|ShgB	|Offset und Invertierung geändert.	
17.08.00	|LeaF	|Freigabe

*)
VAR_INPUT
	x_Enable:BOOL;//Freigabe des Reglers
	f_Ist:REAL;//Istwert
END_VAR
VAR_INPUT PERSISTENT
	x_Invertiert:BOOL;//Bei Kühlfunktionen aktiv
	x_Manuell:BOOL;//Manuelles Regelsignal aktivieren
	f_Sollwert:REAL;//Sollwertvorgabe
	f_Offset:REAL;//Offset
	f_Min:REAL;//Minimales Regelsignal
	f_Max:REAL;//Maximales Regelsignal
	f_Manuell:REAL;//Manuelles Regelsignal
	f_PFaktor:REAL;//Proportionalfaktor
	f_IFaktor:REAL;//Integralfaktor
	t_Takt:timestruct;//Regelungstakt
END_VAR
VAR_OUTPUT
	f_Regelsignal:REAL;//Regelsignal
END_VAR
VAR
	f_IAnteil,f_ISpeicher:REAL;
	f_PAnteil:REAL;
	P_Anteil: PRegler;
	Timer: TON;
	x_Takt:BOOL;
	Timestruct_to_Time:Timestruct_to_Time;
END_VAR

//P Anteil	
	P_Anteil(
		x_Enable:= x_Enable, 
		x_Invertiert:= x_Invertiert, 
		x_Manuell:= FALSE, 
		f_Sollwert:= f_Sollwert, 
		f_Ist:= f_Ist, 
		f_Offset:= f_Offset, 
		f_Min:= -f_Max, 
		f_Max:= f_Max, 
		f_Manuell:= 0, 
		f_PFaktor:= f_PFaktor, 
		f_Regelsignal=> f_PAnteil);

//TImestruct to Time
	Timestruct_to_Time(t_Ein:=t_Takt);
	
//Takt
	Timer(IN:= x_Enable AND NOT x_Takt, PT:= Timestruct_to_Time.t_Aus, Q=> x_Takt, ET=> );
	
//I Anteil
	IF x_Takt AND f_Regelsignal<f_Max AND f_Regelsignal>f_Min THEN
		f_ISpeicher:=f_ISpeicher+f_IFaktor*f_PAnteil;
	END_IF

//Reset Speicher
	IF NOT x_Enable THEN
		f_ISpeicher:=0.0;
	END_IF
	
//Grenzen einhalten	
	f_Regelsignal := LIMIT(f_Min,f_ISpeicher+f_PAnteil,f_Max);
	
//Manuell	
	IF x_Manuell THEN
		f_Regelsignal:=f_Manuell;
	END_IF

END_FUNCTION_BLOCK

// Timer/BLINK_A
(*Wenn x_Ein auf true blinkt der digitale Ausgang in einem asymetrischen Takt, mit den eingegebenen t_BlinkEin und t_BlinkAus Zeiten.
*)
FUNCTION_BLOCK BLINK_A
(*
Versionsverlauf: 
Version		|Autor	|Bemerkung
------------------------------------------------------------------------------------------------------------ 
17.05.00	|KuzR	|erste Freigabe 
17.08.00	|LeaF	|Freigabe

*)
VAR_INPUT
	x_Ein:BOOL;//Eingang Start
END_VAR
VAR_INPUT PERSISTENT
	t_BlinkEin:Timestruct := (wSecond := 5);//Zeiteingabe blinken Ein
	t_BlinkAus:Timestruct := (wSecond := 1);//Zeiteingabe blinken Aus
END_VAR
VAR_OUTPUT
	x_Aus:BOOL;//Digitaler Ausgang
END_VAR
VAR
	Blink:tof;		
	Pause:tof;
	t_PtZeitEIN:TIME;
	t_PtZeitAUS:TIME;
	Timestruct_to_Time: Timestruct_to_Time;
END_VAR

//Wenn Eingang True, dann läuft eingestellte Zeit ab, Ausgang True
	Timestruct_to_Time(t_Ein:=t_BlinkEin , t_Aus=>t_PtZeitEIN );
	Blink(in:=x_Ein AND NOT Pause.Q AND NOT Blink.Q, pt:=t_PtZeitEIN, Q=> x_Aus);

//Pause, läuft eingestellte Zeit ab, Ausgang False
	Timestruct_to_Time(t_Ein:=t_BlinkAus , t_Aus=>t_PtZeitAUS );
	Pause(in:=NOT Pause.Q AND NOT blink.Q, pt:=t_PtZeitAUS);

END_FUNCTION_BLOCK

// Timer/BLINK_S
(*Wenn x_Ein auf true blinkt der digitale Ausgang in einem symetrischen Takt, mit der eingegebenen t_BlinkEin Zeit.
*)
FUNCTION_BLOCK BLINK_S
(*
Versionsverlauf: 
Version		|Autor	|Bemerkung
------------------------------------------------------------------------------------------------------------ 
17.05.00	|KuzR	|erste Freigabe 
17.08.00	|LeaF	|Freigabe

*)
VAR_INPUT
	x_Ein:BOOL;
END_VAR
VAR_INPUT PERSISTENT
	t_BlinkEin:Timestruct := (wSecond := 5);
END_VAR
VAR_OUTPUT
	x_Aus:BOOL;
END_VAR
VAR
	Blink:tof;		
	Pause:tof;
	t_PtZeitEIN:TIME;
	Timestruct_to_Time:Timestruct_to_Time;	
END_VAR

//Wenn Eingang True, dann läuft eingestellte Zeit ab, Ausgang True
	Timestruct_to_Time(t_Ein:=t_BlinkEin, t_Aus=>t_PtZeitEIN );
	Blink(in:=x_Ein AND NOT Pause.Q AND NOT Blink.Q, pt:=t_PtZeitEIN, Q=> x_Aus);

//Pause, Ausgang False
	Timestruct_to_Time(t_Ein:=t_BlinkEin , t_Aus=>t_PtZeitEIN );
	Pause(in:=NOT Pause.Q AND NOT blink.Q, pt:=t_PtZeitEIN);

END_FUNCTION_BLOCK

// Timer/PULSE
(*Ist x_Ein auf true, wird x_Aus auf true gesetzt mit der eingegebenen Ablaufzeit. Sobald x_Ein auf false, dann x_Aus sofort auf false.
*)
FUNCTION_BLOCK PULSE
(*
Versionsverlauf: 
Version		|Autor	|Bemerkung
------------------------------------------------------------------------------------------------------------ 
17.05.00	|KuzR	|erste Freigabe 
17.08.00	|LeaF	|Freigabe

*)
VAR_INPUT
	x_Ein:BOOL;
END_VAR
VAR_INPUT PERSISTENT
	t_Abl:Timestruct := (wSecond := 5);//Eingegebene Ablaufzeit	
END_VAR
VAR_OUTPUT
	x_Aus:BOOL;//Digitaler Ausgang
	t_ET:Timestruct;//Ausgang Ablaufzeit
END_VAR
VAR
	Pulse:tp;
	t_PtZeit:TIME;
	Timestruct_to_Time:Timestruct_to_Time;	
	Time_to_Timestruct: Time_to_Timestruct;
END_VAR

//Wenn Eingang True, dann läuft eingestellte Zeit ab
	Timestruct_to_Time(t_Ein:=t_Abl , t_Aus=>t_PtZeit );
	Pulse(in:=x_Ein, pt:=t_PtZeit,Q=> x_Aus);

//Wenn Eingang False, dann Ausgang sofort auf False
	IF NOT x_Ein THEN
		x_Aus := FALSE;
	END_IF

//Ausgabe Ablaufzeit im timestruct
	Time_to_Timestruct(t_Ein:= Pulse.ET, t_Aus=> t_ET);

END_FUNCTION_BLOCK

// Timer/TOF_Reset
(*TOF Timer der mit einer Reset Funktion erweitert ist.
*)
FUNCTION_BLOCK TOF_Reset
(*
Versionsverlauf: 
Version		|Autor	|Bemerkung
------------------------------------------------------------------------------------------------------------ 
17.06.00	|Shgb	|erste Freigabe 
17.06.01	|ShgB	|Von Time auf Timestruct geändert
17.08.00	|LeaF	|Freigabe

*)
VAR_INPUT
	x_Ein:BOOL;//Eingang
	x_Reset:BOOL;//Ausschaltverzögerung wird auf 0 gesetzt
END_VAR
VAR_INPUT PERSISTENT
	t_time:timestruct := (wMinute := 5);//Ausschaltverzögerung
END_VAR
VAR_OUTPUT
	x_Aus:BOOL;//Ausgang
	t_Restzeit:timestruct;//Restzeit der Timerfunktion
END_VAR
VAR
	Timer: TOF;
	x_ResetFunktion:BOOL;
	Time_to_Timestruct: Time_to_Timestruct;
	Timestruct_to_Time:Timestruct_to_Time;
END_VAR

//Reset
	IF x_Reset THEN
		x_ResetFunktion := TRUE;
	END_IF

	IF x_Ein THEN
		x_ResetFunktion := FALSE;
	END_IF
	
//TImestruct to Time
	Timestruct_to_Time(t_Ein:=t_time);
	
//Beim Ausschalten Timer aktivieren	
	Timer(IN:=x_Ein, PT:= Timestruct_to_Time.t_Aus);

//Restzeit berechnen
	IF NOT x_ResetFunktion THEN
		Time_to_Timestruct(t_Ein:= Timestruct_to_Time.t_Aus-timer.ET, t_Aus=> t_Restzeit);
	ELSE
		Time_to_Timestruct(t_Ein:= T#0S, t_Aus=> t_Restzeit);
	END_IF
	
//Ausgang schalten
	x_Aus:=timer.Q AND NOT x_ResetFunktion;

END_FUNCTION_BLOCK

// Timer/TON_Reset
(*TON Timer der mit einer Reset Funktion erweitert ist.
*)
FUNCTION_BLOCK TON_Reset
(*
Versionsverlauf: 
Version		|Autor	|Bemerkung
------------------------------------------------------------------------------------------------------------ 
17.06.00	|Shgb	|erste Freigabe 
17.08.00	|LeaF	|Freigabe

*)
VAR_INPUT
	x_Ein:BOOL;//Eingang
	x_Reset:BOOL;//Einschaltverzögerung wird auf 0 gesetzt
END_VAR
VAR_INPUT PERSISTENT
	t_time:timestruct := (wMinute := 5);//Ausschaltverzögerung
END_VAR
VAR_OUTPUT
	x_Aus:BOOL;//Ausgang
	t_Restzeit:timestruct;//Restzeit der Timerfunktion
END_VAR
VAR
	Timer: TON;
	x_Timer,x_ResetFunktion:BOOL;
	t_ET:TIME;
	Time_to_Timestruct: Time_to_Timestruct;
	Timestruct_to_Time:Timestruct_to_Time;
END_VAR

//Reset
	IF x_Reset THEN
		x_ResetFunktion := TRUE;
	END_IF

	IF NOT x_Ein THEN
		x_ResetFunktion := FALSE;
	END_IF
	
//TImestruct to Time
	Timestruct_to_Time(t_Ein:=t_time);
	
//Beim Einschalten Timer aktivieren	
	Timer(IN:= x_Ein, PT:= Timestruct_to_Time.t_Aus, Q=> x_timer, ET=> t_ET);

//Restzeit berechnen
	IF NOT x_ResetFunktion THEN
		Time_to_Timestruct(t_Ein:= Timestruct_to_Time.t_Aus-t_ET, t_Aus=> t_Restzeit);
	ELSE
		Time_to_Timestruct(t_Ein:= T#0S, t_Aus=> t_Restzeit);
	END_IF
	
//Ausgang schalten
	x_Aus:= x_timer OR x_ResetFunktion;

END_FUNCTION_BLOCK

// Timer/Work
(*Betriebstunden- und Impulszäheler
*)
FUNCTION_BLOCK Work
(*
Versionsverlauf: 
Version		|Autor	|Bemerkung
------------------------------------------------------------------------------------------------------------ 
17.06.00	|Shgb	|erste Freigabe 
17.08.00	|ShgB	|Betriebsstunden nicht mit DT berechnet da Time Format nur bis 49 Tage geht.

*)
VAR_INPUT
	x_Ein:BOOL;//Eingang
	x_Reset:BOOL;//Stellt die Zähler auf 0 zurück
END_VAR
VAR_INPUT PERSISTENT
	t_StartBetriebsstunden:TIMESTRUCT;//Betriebsstunden die bei einem Reset auf den Ausgang geschrieben werden
	i_StartEinschaltungen:INT;//Anzahl Einschaltungen die bei einem Reset auf den Ausgang geschriben werden
END_VAR
VAR_OUTPUT PERSISTENT
	t_Betriebsstunden:TIMESTRUCT;//Anzeige der bis jetzt geleisteten Betriebsstunden
	i_Einschaltungen:INT;//Anzeige Einschaltimpulse
END_VAR
VAR
	x_Speicher: BOOL;
	w_Speicher:WORD;
END_VAR

//Impulse zählen
	IF x_Ein AND NOT x_Speicher THEN
		i_Einschaltungen:= i_Einschaltungen+1;
	END_IF
	x_Speicher:=x_Ein;
	
//Betriebsstundenzähler
	IF x_Ein THEN
		IF w_Speicher <> Globale_Uhr.systemtimestruct.wSecond THEN
			t_Betriebsstunden.wSecond := t_Betriebsstunden.wSecond +1;
			IF t_Betriebsstunden.wSecond>=60 THEN
				t_Betriebsstunden.wSecond:=0;
				t_Betriebsstunden.wMinute:=t_Betriebsstunden.wMinute+1;
				IF t_Betriebsstunden.wMinute>=60 THEN
					t_Betriebsstunden.wMinute:=0;
					t_Betriebsstunden.wHour:=t_Betriebsstunden.wHour+1;
					IF t_Betriebsstunden.wHour >=24 THEN
						t_Betriebsstunden.wHour:=0;
						t_Betriebsstunden.wDay:=t_Betriebsstunden.wDay+1;						
					END_IF
				END_IF
			END_IF
			w_Speicher:=Globale_Uhr.systemtimestruct.wSecond;
		END_IF
	END_IF	

//Reset
	IF x_Reset THEN
		i_Einschaltungen:=i_StartEinschaltungen;
		t_Betriebsstunden:=t_StartBetriebsstunden;
	END_IF

END_FUNCTION_BLOCK

